(* CoDeSys 2.3 project: esx_ioxp_PPS_load_16.pro *)
(* Libraries: esx_ioxp.lib 19.12.13 13:14:40, Util.lib 18.5.10 15:14:28, Standard.lib 4.10.05 11:14:46 *)

(* PLC configuration (modules and I/O channels)
gq_Ignition AT %IX0.0 [X_SYS_IGNITION] Ignition pin (D+)
gs16_TempBoard AT %IW1 [X_SYS_TEMP_BOARD] System temperature in degree Celsius
gu32_TimeMs AT %ID1 [X_SYS_TIME_MS] System time in ms
gq_StayAlive AT %QX0.0 [X_SYS_STAY_ALIVE] Stay alive mechanism
gq_Relay AT %QX1.0 [X_SYS_RELAY_1] Safety relay
gs32_SensorSupply AT %QD1 [X_SYS_SENSOR_SUPPLY_1] External sensor supply
gs32_IO01 AT %QD2 [InOut] --- Inj 2-1 ----IO01, PIN 9 (PWM H/L, DO, CC, VIN (40V), DIN) {InOut_Type = X_OUT_TYPE_DIGITAL; InOut_FilterConfig = 0; InOut_Circuit1 = X_OUT_CIRCUIT_HIGH_SIDE; InOut_Circuit2 = X_IN_CIRCUIT_NO_PULL_UP; PWM_MaxValue = 10000}
gs32_IO02 AT %QD3 [InOut] ---- Inj 2-2 ---- IO02, PIN 8 (PWM H/L, DO, CC, VIN (40V), DIN) {InOut_Type = X_IN_TYPE_VOLTAGE_40V; InOut_FilterConfig = 0; InOut_Circuit1 = X_IN_CIRCUIT_ACTIVE_HIGH; InOut_Circuit2 = X_IN_CIRCUIT_PULL_UP; PWM_MaxValue = 10000}
gs32_IO03 AT %QD4 [InOut] --- GAS LED BAR  ---  IO03, PIN 7 (PWM H/L, DO, CC, VIN ( {InOut_Type = X_OUT_TYPE_PWM; InOut_FilterConfig = 0; InOut_Circuit1 = X_OUT_CIRCUIT_PUSH_PULL; InOut_Circuit2 = X_IN_CIRCUIT_NO_PULL_UP; PWM_MaxValue = 10000}
gs32_IO04 AT %QD5 [InOut] --- PPS_emul---- IO04, PIN 6 (PWM H/L, DO, CC, VIN (40V), DIN) {InOut_Type = X_OUT_TYPE_PWM; InOut_FilterConfig = 0; InOut_Circuit1 = X_OUT_CIRCUIT_HIGH_SIDE; InOut_Circuit2 = X_IN_CIRCUIT_NO_PULL_UP; PWM_MaxValue = 10000}
gs32_IO05 AT %QD6 [InOut] -----Inj 1-2 ----- IO05, PIN 13 (PWM H, DO, DIN) {InOut_Type = X_OUT_TYPE_DIGITAL; InOut_FilterConfig = 0; InOut_Circuit1 = X_OUT_CIRCUIT_HIGH_SIDE; InOut_Circuit2 = X_IN_CIRCUIT_NO_PULL_UP; PWM_MaxValue = 10000}
gs32_IO06 AT %QD7 [InOut] ---Inj1-1--- IO06, PIN 12 (PWM H, DO, DIN) {InOut_Type = X_OUT_TYPE_DIGITAL; InOut_FilterConfig = 0; InOut_Circuit1 = X_OUT_CIRCUIT_HIGH_SIDE; InOut_Circuit2 = X_IN_CIRCUIT_NO_PULL_UP; PWM_MaxValue = 10000}
gs32_IO07 AT %QD8 [InOut] --- Inj3-1 -----IO07, PIN 11 (PWM H, DO, DIN) {InOut_Type = uninitialized; InOut_FilterConfig = 0; InOut_Circuit1 = X_IN_CIRCUIT_ACTIVE_HIGH; InOut_Circuit2 = X_IN_CIRCUIT_NO_PULL_UP; PWM_MaxValue = 10000}
gs32_IO08 AT %QD9 [InOut] --- Inj 3-2 --  IO08, PIN 10 (PWM H, DO, DIN) {InOut_Type = X_OUT_TYPE_DIGITAL; InOut_FilterConfig = 0; InOut_Circuit1 = X_OUT_CIRCUIT_HIGH_SIDE; InOut_Circuit2 = X_IN_CIRCUIT_NO_PULL_UP; PWM_MaxValue = 10000}
gs32_IO09 AT %ID2 [InOut] --- SPEED --- IO09, PIN 2 (DIN, FIN, IIN) {InOut_Type = X_IN_TYPE_FREQUENCY; InOut_FilterConfig = 0; InOut_Circuit1 = X_OUT_CIRCUIT_HIGH_SIDE; InOut_Circuit2 = X_IN_CIRCUIT_NO_PULL_UP; PWM_MaxValue = 10000}
gs32_IO10 AT %ID3 [InOut] ---RPM--- IO10, PIN 3 (DIN, FIN, IIN) {InOut_Type = X_IN_TYPE_FREQUENCY; InOut_FilterConfig = 0; InOut_Circuit1 = X_IN_CIRCUIT_ACTIVE_HIGH; InOut_Circuit2 = X_IN_CIRCUIT_NO_PULL_UP; PWM_MaxValue = 10000}
gs32_IO11 AT %ID4 [InOut] IO11, PIN 4 (DIN, FIN, IIN) {InOut_Type = uninitialized; InOut_FilterConfig = 0; InOut_Circuit1 = X_IN_CIRCUIT_ACTIVE_HIGH; InOut_Circuit2 = X_IN_CIRCUIT_NO_PULL_UP; PWM_MaxValue = 10000}
gs32_IO12 AT %ID5 [InOut] ---BLOCK ON--- IO12, PIN 5 (DIN) {InOut_Type = X_IN_TYPE_VOLTAGE_10V; InOut_FilterConfig = 0; InOut_Circuit1 = X_IN_CIRCUIT_ACTIVE_HIGH; InOut_Circuit2 = X_IN_CIRCUIT_NO_PULL_UP; PWM_MaxValue = 10000}
gs32_IO13 AT %ID6 [InOut] IO13, PIN 38 (CIN (20mA), DIN) {InOut_Type = uninitialized; InOut_FilterConfig = 0; InOut_Circuit1 = X_IN_CIRCUIT_ACTIVE_HIGH; InOut_Circuit2 = X_IN_CIRCUIT_NO_PULL_UP; PWM_MaxValue = 10000}
gs32_IO14 AT %ID7 [InOut] IIO14, PIN 24 (CIN (20mA), DIN) {InOut_Type = uninitialized; InOut_FilterConfig = 0; InOut_Circuit1 = X_IN_CIRCUIT_ACTIVE_HIGH; InOut_Circuit2 = X_IN_CIRCUIT_NO_PULL_UP; PWM_MaxValue = 20000}
gs32_IO15 AT %ID8 [InOut] - Injecor temp ----IO15, PIN 39 (CIN (20mA), DIN) {InOut_Type = X_IN_TYPE_CURRENT; InOut_FilterConfig = 0; InOut_Circuit1 = X_IN_CIRCUIT_ACTIVE_HIGH; InOut_Circuit2 = X_IN_CIRCUIT_NO_PULL_UP; PWM_MaxValue = 4000000}
gs32_IO16 AT %ID9 [InOut] IO16, PIN 25 (CIN (20mA), DIN) {InOut_Type = uninitialized; InOut_FilterConfig = 0; InOut_Circuit1 = X_IN_CIRCUIT_ACTIVE_HIGH; InOut_Circuit2 = X_IN_CIRCUIT_NO_PULL_UP; PWM_MaxValue = 10000}
gs32_IO17 AT %ID10 [InOut] IO17, PIN 40 (CIN (20mA), DIN) {InOut_Type = uninitialized; InOut_FilterConfig = 0; InOut_Circuit1 = X_IN_CIRCUIT_ACTIVE_HIGH; InOut_Circuit2 = X_IN_CIRCUIT_NO_PULL_UP; PWM_MaxValue = 10000}
gs32_IO18 AT %ID11 [InOut] ----- SOLARKA meter ----- IO18, PIN 26 (CIN (20mA), DIN) {InOut_Type = X_IN_TYPE_CURRENT; InOut_FilterConfig = 0; InOut_Circuit1 = X_IN_CIRCUIT_ACTIVE_HIGH; InOut_Circuit2 = X_IN_CIRCUIT_NO_PULL_UP; PWM_MaxValue = 20000}
gs32_IO19 AT %ID12 [InOut] --- GAS meter  ----- IO19, PIN 41 (CIN (20mA), DIN) {InOut_Type = X_IN_TYPE_CURRENT; InOut_FilterConfig = 0; InOut_Circuit1 = X_IN_CIRCUIT_ACTIVE_HIGH; InOut_Circuit2 = X_IN_CIRCUIT_NO_PULL_UP; PWM_MaxValue = 10000}
gs32_IO20 AT %ID13 [InOut] ---Reductor_temp---  IO20, PIN 27 (CIN (20mA), DIN) {InOut_Type = X_IN_TYPE_CURRENT; InOut_FilterConfig = 0; InOut_Circuit1 = X_IN_CIRCUIT_ACTIVE_HIGH; InOut_Circuit2 = X_IN_CIRCUIT_NO_PULL_UP; PWM_MaxValue = 20000}
gs32_IO21 AT %ID14 [InOut] ---Turbo_pressure--- IO21, PIN 34 (VIN (10V), DIN) {InOut_Type = X_IN_TYPE_VOLTAGE_10V; InOut_FilterConfig = 0; InOut_Circuit1 = X_IN_CIRCUIT_ACTIVE_HIGH; InOut_Circuit2 = X_IN_CIRCUIT_NO_PULL_UP; PWM_MaxValue = 10000}
gs32_IO22 AT %ID15 [InOut] ---Reductor_press---   IO22, PIN 20 (VIN (10V), DIN) {InOut_Type = X_IN_TYPE_VOLTAGE_10V; InOut_FilterConfig = 0; InOut_Circuit1 = X_IN_CIRCUIT_ACTIVE_HIGH; InOut_Circuit2 = X_IN_CIRCUIT_NO_PULL_UP; PWM_MaxValue = 10000}
gs32_IO23 AT %ID16 [InOut] --- EGT ----IO23, PIN 35 (VIN (10V), DIN) {InOut_Type = X_IN_TYPE_VOLTAGE_10V; InOut_FilterConfig = 0; InOut_Circuit1 = X_IN_CIRCUIT_ACTIVE_HIGH; InOut_Circuit2 = X_IN_CIRCUIT_NO_PULL_UP; PWM_MaxValue = 10000}
gs32_IO24 AT %ID17 [InOut] ---PPS1--- IO24, PIN 21 (VIN (10V), DIN) {InOut_Type = X_IN_TYPE_VOLTAGE_10V; InOut_FilterConfig = 0; InOut_Circuit1 = X_IN_CIRCUIT_ACTIVE_HIGH; InOut_Circuit2 = X_IN_CIRCUIT_NO_PULL_UP; PWM_MaxValue = 10000}
gs32_IO25 AT %ID18 [InOut] --- PPS2 ---- IO25, PIN 36 (VIN (10V), DIN) {InOut_Type = X_IN_TYPE_VOLTAGE_10V; InOut_FilterConfig = 0; InOut_Circuit1 = X_IN_CIRCUIT_ACTIVE_HIGH; InOut_Circuit2 = X_IN_CIRCUIT_NO_PULL_UP; PWM_MaxValue = 10000}
gs32_IO26 AT %ID19 [InOut] ---- Check_PPS_emul ----O26, PIN 22 (VIN (10V), DIN) {InOut_Type = X_IN_TYPE_VOLTAGE_10V; InOut_FilterConfig = 0; InOut_Circuit1 = X_IN_CIRCUIT_ACTIVE_LOW; InOut_Circuit2 = X_IN_CIRCUIT_NO_PULL_UP; PWM_MaxValue = 5000}
RS232 [X_SER_1] node 1, in %IB80 out %QB40 {X_SER_BITRATE = 19200; X_SER_STOPBITS = 1; X_SER_MODE = 8 data bits - no parity; X_SER_RX_BUFSIZE = 256; X_SER_TX_BUFSIZE = 256}
CAN1 [X_CAN_BUS_1_XC2] node 2, in %IB80 out %QB40 {X_CAN_BUS_BITRATE = 125000; X_CAN_BUS_11BIT_MASK = 16#7FF; X_CAN_BUS_29BIT_MASK = 16#1FFFFFFF}
TX AT %ID20 [X_CAN_OBJ_HANDLE] CAN object handle
CAN RX Object [X_CAN_OBJ_RX_XC2] node 11770, in %IB84 out %QB40 {X_CAN_OBJ_ID = 16#100; X_CAN_OBJ_XTD = 11bit; X_CAN_OBJ_MASK = 16#7FF; X_CAN_OBJ_SOFT_BUFFER = 10; X_CAN_OBJ_HARD_BUFFER = 10}
  RX AT %ID21 [X_CAN_OBJ_HANDLE] CAN object handle
CAN2 [X_CAN_BUS_2_XC2] node 3, in %IB80 out %QB40 {X_CAN_BUS_BITRATE = 125000; X_CAN_BUS_11BIT_MASK = 16#7FF; X_CAN_BUS_29BIT_MASK = 16#1FFFFFFF}
*)

(* Task configuration *)
TASK Get_RPM (PRIORITY := 3, INTERVAL := T#300ms);
	Get_RPM_speed();
	Get_EGT();
END_TASK
TASK Main (PRIORITY := 20, INTERVAL := T#100ms);
	PLC_PRG();
	DFPRS_Change_Cal_Table();
	Get_Currents();
	Get_Reductor_press();
END_TASK
TASK Act_control (PRIORITY := 2, INTERVAL := T#100ms);
	Act_control();
END_TASK
TASK Get_turbo (PRIORITY := 3, INTERVAL := T#50ms);
	Get_Turbo();
END_TASK
TASK Get_key (PRIORITY := 10, INTERVAL := T#50ms);
	Get_Key();
END_TASK
TASK Get_low_freq (PRIORITY := 5, INTERVAL := T#300ms);
	Get_Gas_meter();
	Get_Reductor_temp();
	Get_Inj_temp();
	Get_FUEL_meter();
	Get_cPPS();
END_TASK
TASK CAN (PRIORITY := 20, INTERVAL := T#50ms);
	Send();
	Recieve();
END_TASK

(* Global variable list: Global_Constant *)
VAR_GLOBAL CONSTANT
(********************** Разное ***************************************************************************)

	TOOTH_NUM					:WORD:=58;				(* Количество зубцов на коленвале *)
	Min_time_cnange_mode_EGT:UDINT:=60000; 		(* Минимальное время в мс между сменами режимов ГАЗ и ДИЗЕЛЬ для обновления статистических значений EGT *)
	Inj_PWM_period				:WORD:=250;				(* Период работы форсунок HANA=16 HZ задается в кол-ве рабочих циклов по 250 мкс*)

(******************** Настойки системы безопасности **********************************)

	RPM_count:WORD:=10;						(* Максимальное количество циклов неправильного RPM, когда считаем это флуктуацией *)
	PPS_err_time:WORD:=3;					(* Максимальное количество циклов неправильного PPS, когда считаем это флуктуацией *)
	Min_Reductor_press_time:WORD:=10;	(* Макстмально допустимое время минимального давления *)
	Reductor_temp_err_time:WORD:=100;	(* Через столько циклов блок опять включится что бы проверить температуру редуктора после первого включения по превышению *)
	EGT_err_time:WORD:=100;					(* Через столько циклов блок опять включится что бы проверить EGT после отключения по превышению EGT *)
	Max_inj_current_time:BYTE:=100;		(* Макстмально допустимое время протекания максимального тока через форсунку в РАБОЧИХ циклах подпрограммы *)

END_VAR

(* Global variable list: Global_Variables *)
VAR_GLOBAL

	(* Значения считывемые с входов контролера *)

	RPM						:WORD; 				(* RPM *)
	Turbo_pressure	      :DINT;				(* Turbo pressure in mV *)
	PPS1	      			:DINT;				(* Основная педаль газа in mV *)
	OLD_PPS					:DINT;
	PPS2						:DINT;				(* Дублирующая педаль газа *)
	EGT						:DINT;				(* Температуры выхлопных газов *)
	Reductor_temp			:DINT;				(* Температура редуктора *)
	Reductor_press			:DINT;				(* Давление после редуктора *)
	Gas_meter				:DINT;				(* Давление газа *)
	Injector_temp			:DINT;				(* Температура инжекторов *)
	FUEL_meter				:DINT;				(* Значение датчика солярки *)
	Speed						:DINT;				(* Счетчик импульсов коленвала *)


	(* РАЗНОЕ *)
	Inj_PWM_time			:BYTE;	 			(* Длительность холдового PWM для газового инжектора, расчитывается исходя из данных калибровки в циклах по 250 мкс*)
	HOLD_time				:BYTE;
	Turn_start				:UDINT;				(* Системное время когда была нажата кнопка управления *)
	Count_min_reductor_press:WORD;			(* Счетчик времени для определения подлинного события падения давления в редукторе *)
	PPS1_emul				:DINT;				(* Уровень PWM для эмулирования первой педали газа *)
	cPPS1_emul				:DINT;				(* Уровень ФАКТИЧЕСКОГО измеренного напряжения эмуляции PPS *)
	FUEL_volume				:REAL;				(* Объем топлива в литрах *)
	Load						:BYTE;				(* Отношение импульсов датчика распредвала и коленвала *)

	(* Значения тока протекающего через Пин, подключеннный к форсунке. 2 Пина = 1 форсунка *)

	s32_Current_Inj1_1			: DINT;
	s32_Current_Inj1_2			: DINT;
	s32_Current_Inj2_1			: DINT;
	s32_Current_Inj2_2			: DINT;
	s32_Current_Inj3_1			: DINT;
	s32_Current_Inj3_2			: DINT;

	(* Структуры данных для записи в EEPROM *)

	p							:Parameters;		(* Сруктура с настройками, при старте контролера подгружаться из EEPROM*)
	a							:Always_write;		(* Структура тоже с настройками. но которая ВСЕГДА при записывается EEPROM при выключении  *)

	(* Логические переменные для включения различных режимов *)

	Flag_ECU_ON				:BOOL;				(* Контроллер включен *)
	Flag_PWM_researh		:BOOL;				(* Включения режима исследования отношения PWM к выходу операционного усилителя *)
	Flag_Inj_PWM_cor		:BOOL;				(* Показывает что была произведена коррекци Inj_PWM по превышению предельных значений *)
	Flag_first_start		:BOOL:=TRUE;		(* Первое включение, для проверки давления *)
	Flag_24V					:BOOL:=FALSE;   	(* 24 Вольтовое газовое оборудоыание, нужен для уменьшения подачи через спецкоды *)

	(* Индивидуальное включение/выключение форсунок *)
	(* Скания все три включены *)
	(* Газель включен первый канал , 2 форсунки. 2 и 3 - выключены  *)
	Flag_Inj1_ON			:BOOL:=TRUE;
	Flag_Inj2_ON			:BOOL:=FALSE;
	Flag_Inj3_ON			:BOOL:=FALSE;

	(* Режим тестирования работы газовых инжекторов *)
	Flag_test_inj: BOOL;

	(* Логические переменные, использующиеся для обмена по CAN калибровками с питоновской прграммой *)

	Flag_CAN_send			:BOOL;				(* Запрос по CAN на посылку калибровки *)
	Flag_CAN_recieve		:BOOL;				(* Запрос по CAN на прием калибровки *)
	Flag_CAN					:BOOL;				(* Режим обмена по CAN калибровками активирован *)
	Flag_CAN_data			:BOOL;
	Flag_CAN_CRC16			:BOOL;
	Flag_CAN_Write			:BOOL;


	(*********** Флаги ошибок  *****************************)

	Err_RPM					:BOOL;				(* RPM более чем RPM_count циклов не в пределах RPM_min - RPM_max *)
	Err_EGT					:BOOL;				(* Превышен максимальный уровень EGT *)
	Err_Reductor_temp		:BOOL;				(* Недостигнута рабочая температура редуктора *)
	Err_Inj1					:BOOL;				(* Долговременно превышен максимальный ток в инжекторе 1 *)
	Err_Inj2					:BOOL;				(* Долговременно превышен максимальный ток в инжекторе 2 *)
	Err_Inj3					:BOOL;				(* Долговременно превышен максимальный ток в инжекторе 3 *)
	Err_Inj_temp			:BOOL;				(* Превышение температуры инжекторов *)
	Err_Reductor_press	:BOOL;				(* Давление в редукторе ниже нормы *)
	Err_PPS					:BOOL;				(* PPS ниже или выше допустимого значения *)

	Can_buffer				:ARRAY [1..6000] OF BYTE; 											(* Буфер для сохранения области EEPROM 750*8 *)

END_VAR

(* Data type *)
(* Эта структурв перезаписывается каждый раз при выключении *)

TYPE Always_write :
STRUCT
		Flag_byte					:BYTE;				(* 8 флагов, для хранения в EEPROM *)
		EGT_max_abs_GAS			:DINT;				(* Абсолютное максимальное достигнутое значение EGT за все время работы контроллера на ГАЗУ *)
		EGT_max_abs_DIESEL		:DINT;				(* Абсолютное максимальное достигнутое значение EGT за все время работы контроллера на ДИЗЕЛЕ *)
		EGT_max_sessions_GAS		:DINT;				(* Абсолютное максимальное значение EGT за прошлую сессию на ДИЗЕЛЕ *)
		EGT_max_sessions_DIESEL	:DINT;				(* Абсолютное максимальное значение EGT за прошлую сессию на ГАЗУ *)
END_STRUCT
END_TYPE

(* Data type *)
TYPE Cal_data :
STRUCT
	Gas: BYTE;
	Diesel: BYTE;
END_STRUCT
END_TYPE

(* Data type *)
(* Используется для обхода ограничений по редактированию таблиц в визуализации *)

TYPE FLS :
STRUCT
	a:WORD;
END_STRUCT
END_TYPE

(* Data type *)
(* Структура данных, хранящаяся в EEPROM *)
TYPE Parameters :
	STRUCT
		(* Таблица для 3-х мерной калибровки подачи газа и дизеля. Оброты, надув, педаль ( разносится автоматически ) *)
		Cal_table					:ARRAY [1..16,1..16] OF Cal_data;
		(* Основные таблицы границ  - обротов, надува и педали газа *)
		RPM_table					:ARRAY[1..16] OF WORD;	(* Значения RPM *)
		Turbo_table					:ARRAY[1..16] OF WORD;	(* Значения наддува турбины *)
		PPS_table					:ARRAY[1..16] OF WORD;	(* Значения нажатия на педаль газа *)
		PPS1_emul_PWM				:ARRAY[1..32] OF WORD;	(* Соответствие значения эмуляции и частотв PWM *)
		(* Учет топлива *)
		LED_BAR_PWM					:ARRAY[1..5]  OF WORD;	(* Соответствие PWM каждому диапазону датчика давления для индикатора *)
		Gas_meter_volume			:ARRAY[1..5]  OF DINT;	(* Разбивка датчика давления в баллоне на диапазоны *)
		FUEL_meter_dat				:ARRAY[1..32] OF WORD;	(* Калибровка датчика солярки, соответствие показаний физическому объему, показания датчика *)
		FUEL_meter_liter			:ARRAY[1..32] OF WORD;	(* Калибровка датчика литры *)
		(******************** Настойки системы безопасности **********************************)
		EGT_max						:WORD;						(* Максимально допустимый уровень EGT *)
		(*********** Пределы допустимых значений RPM ******************************)
		RPM_Min						:WORD;						(* Минимальный порог допкстимого RPM *)
		RPM_Max						:WORD;						(* Максимальный порог допустимого RPM *)
		(*********** Пределы допустимых для редуктора ******************************)
		Reductor_temp_work		:WORD;						(* Минимальная температура редуктора для включения блока *)
		Min_Reductor_press		:WORD;						(* Минимальное давление редуктора для включения блока *)
		(*********** Пределы допустимых для педали газа ******************************)
		PPS1_min						:WORD;						(* Минимальный порог для PPS *)
		PPS1_max						:WORD;						(* Максимальный порог для PPS *)
		PPS2_min						:WORD;						(* Минимальный порог для PPS *)
		PPS2_max						:WORD;						(* Максимальный порог для PPS *)
		PPS_ratio_min				:REAL;						(* Минимальный корректный порог соотношений значений PPS1 и PPS2 *)
		PPS_ratio_max				:REAL;						(* Максимальный корректный порог соотношений значений PPS1 и PPS2 *)
		(**************** Управление форсунками ***************************************************************************)
		Inj_Low_period				:WORD;						(* Задание скважности PWM форсунок (соотношение кол-ва ЦИКЛОВ низкого сигнала к одному ВЫСОКОМУ циклу), подбирается имперически по условию соблюдения уровня холдового тока на форсунке *)
		Inj_High_period			:WORD;						(* Задание скважности PWM форсунок (соотношение кол-ва ЦИКЛОВ низкого сигнала к одному ВЫСОКОМУ циклу), подбирается имперически по условию соблюдения уровня холдового тока на форсунке *)
		Inj_MAX_hold_time			:BYTE;						(* В циклах по 250 мкс !Максимально возможная длительность холда для форсунок на больших нагрузках *)
		Inj_MAX_hold_time_min	:BYTE;						(* Максимально возможная длительность холда для форсунок на малых нагрузках *)
		Inj_peak_curent_cycle	:BYTE;						(* Количество срабатываний цикла обработчика прерываний, для генерирования импульса длительности открытия форсунки с пиковым током в циклах по 250 мкс*)
		(* SCANIA P380 -  Максимальная температура форсунок 90 C при балластном резисторе 1050 Ом  4325 *)
		(* Газель - Максимальная температура форсунок 110 C при балластном резисторе 560 Ом* это 16000, но так как температура растет очень медленно то для подстраховки ставим 14000*)
		Inj_temp_max				:DINT;
		Max_inj_current			:DWORD;						(* Максимальный длительный ток через газовые форсунки в микроамперах *)
		Min_inj_current			:DWORD;						(* Минимальный длительный ток ( обрыв ) через газовые форсунки в микроамперах *)

		Speed_limit					:WORD;						(* Минимальная скорость с какой начинать подачу газа и эмуляцию *)
		Load_table					:ARRAY[1..16] OF WORD;	(* Значения нажатия на педаль газа *)
		GAS_Load_table				:ARRAY[1..16] OF INT;	(* Значения нажатия на педаль газа *)
		DIESEL_Load_table			:ARRAY[1..16] OF INT;	(* Значения нажатия на педаль газа *)
	END_STRUCT
END_TYPE

(* POU Ввод данных/Get_RPM_speed, ST *)
PROGRAM Get_RPM_speed
VAR

	s16_Return   		: INT;
   Old_pulse_counter, Pulse_counter,s32_Counter    	: DINT; (* Набор переменных для вычисления RPM *)
	Old_pulse_counter_speed,s32_Counter_speed    	: DINT; (* Набор переменных для вычисления оборотов коленвала *)
   fb_InGetCounter   : FB_x_in_get_counter;

	cycle_time: DINT;
	old_time: DINT;
	Flag_speed_OK:BOOL;				(* Флаг для визуализации *)
	i: WORD:=RPM_count;			(* Для начала работы нужно хоть одно правильное значение RPM *)
END_VAR
(* Получаем количество импульсов ( импульс=2 сигнала=открывающий и закрывающий фронт )с датчика Холла *)
fb_InGetCounter(ou16_Channel:=X_IN_10, os32_Value=>s32_Counter, os16_Status=>s16_Return);
(* Вычисляем количество импульсов за цикл работы этой прграммы *)
Pulse_counter:=s32_Counter-old_pulse_counter;
Old_pulse_counter:=s32_Counter;
(* Вычисляем время цикла в ms*)
cycle_time:=gu32_TimeMs-old_time;
old_time:=gu32_TimeMs;
(* Переводим в RPM с учетом отсутствующих зубов и времени цикла 30000=1000*60/2 *)
RPM:=DINT_TO_WORD((Pulse_counter*30000/cycle_time)/TOOTH_NUM);
Check_RPM();

(* Получаем количество импульсов ( импульс=2 сигнала=открывающий и закрывающий фронт )с датчика Холла *)
fb_InGetCounter(ou16_Channel:=X_IN_09, os32_Value=>s32_Counter_speed, os16_Status=>s16_Return);
(* Вычисляем количество импульсов за цикл работы этой прграммы *)
Speed:=s32_Counter_speed-old_pulse_counter_speed;
Old_pulse_counter_speed:=s32_Counter_speed;
(* Соотношение между оборотами двигателя и оборотами коленвала *)
IF Speed <> 0 THEN
	Load:=DINT_TO_BYTE(Pulse_counter/Speed);
ELSE
	Load:=0;
END_IF
(* Для визуализации *)
IF speed > p.Speed_limit THEN
	Flag_speed_OK:=TRUE;
ELSE
	Flag_speed_OK:=FALSE;
END_IF
END_PROGRAM
ACTION Check_RPM:
(* Находится ли RPM в допустимых пределах ? *)
IF RPM < p.RPM_min OR RPM > p.RPM_max THEN
	i:=i+1;
ELSE
	i:=0;
END_IF
(* Если RPM выходит задопустимые пределы RPM_count раз подряд, тогда ошибка *)
IF i>=RPM_count THEN
	Err_RPM:=TRUE;
	i:=RPM_count;					(* Что бы избежать переполнения и ложного сброса флага *)
ELSE
	Err_RPM:=FALSE;
END_IF
END_ACTION

(* POU Ввод данных/Get_EGT, ST *)
PROGRAM Get_EGT
VAR
	fb_InGetValue   : FB_x_in_get_value;
	s16_Return      : INT;
	EGT_err_flag: BOOL; (* EGT уже больше, но пока время для установления главного флага еще не вышло *)
	Count_max_EGT: WORD;
	Flag_EGT_reset: BOOL;
END_VAR
fb_InGetValue(ou16_Channel:=X_IN_23, os32_Value=>EGT, os16_Status=>s16_Return);

(* Если EGT превысило допустимую температуру, то следующий контроль EGT на возможное включение блока произойдет через некоторое время *)

IF EGT_err_flag AND  Count_max_EGT < EGT_err_time THEN
	Count_max_EGT:=Count_max_EGT+1;
ELSE
	Count_max_EGT:=0;
	(* Находится ли EGT в допустимых пределах ? *)
	IF EGT > p.EGT_max THEN
		EGT_err_flag:=TRUE;
		Err_EGT:=TRUE;
	ELSE
		EGT_err_flag:=FALSE;
		Err_EGT:=FALSE;
	END_IF
END_IF

(* Контроль, что бы между сменами режимов прошло достаточно кол-ва времени *)
IF (gu32_TimeMs-Turn_start) > Min_time_cnange_mode_EGT THEN
(* Запись максимального значения EGT в как течении сесии так и абсолютно за все время *)
		IF Flag_ECU_ON THEN
				IF EGT > a.EGT_max_sessions_GAS	THEN
					a.EGT_max_sessions_GAS:=EGT;
				END_IF
				IF EGT > a.EGT_max_abs_GAS	THEN
					a.EGT_max_abs_GAS:=EGT;
				END_IF
		ELSE
				IF EGT > a.EGT_max_sessions_DIESEL	THEN
					a.EGT_max_sessions_DIESEL:=EGT;
				END_IF
				IF EGT > a.EGT_max_abs_DIESEL	THEN
					a.EGT_max_abs_DIESEL:=EGT;
				END_IF
		END_IF
END_IF

(* Если нажата кнопка RESET в визуализации, то сбрасываем все значения в структуре always_write где хранятся байт флагов и значения EGT *)
IF Flag_EGT_reset THEN
	a.EGT_max_abs_GAS:=0;
	a.EGT_max_abs_DIESEL:=0;
	a.EGT_max_sessions_GAS:=0;
	a.EGT_max_sessions_DIESEL:=0;
	Flag_EGT_reset:=FALSE;
END_IF
END_PROGRAM

(* POU PLC_PRG, ST *)
PROGRAM PLC_PRG
VAR
	q_FirstCycle	: BOOL := TRUE;

	fb_SysClose		: FB_x_sys_close;
	fb_SsvTrigger	: FB_x_ssv_trigger;
	s16_Return,s16_Return3		: INT;

(*  Работа с входами *)
	fb_InInit    	: FB_x_in_init;
(* Работы с выходами *)
	fb_OutInit  	: FB_x_out_init;
	fb_OutSetFrequency   : FB_x_out_set_frequency;
	fb_OutSetValue   : FB_x_out_set_value;
(* Работа с таймером *)
   fb_TimClose   : FB_x_tim_close;
   fb_TimInit    : FB_x_tim_init;
   fb_TimSet     : FB_x_tim_set;
(* Работа с энергонезависимой памятью *)
	fb_EepWrite   	: FB_x_eep_write;
	fb_EepRead  	: FB_x_eep_read;

	i,k,z								:BYTE;				(* Служат для формирования байта флагов *)

	EGT_max_prev_sessions_GAS		:DINT;				(* Абсолютное максимальное значение EGT за прошлую сессию на ДИЗЕЛЕ *)
	EGT_max_prev_sessions_DIESEL	:DINT;				(* Абсолютное максимальное значение EGT за прошлую сессию на ГАЗУ *)

	Count_off: BYTE;
END_VAR
IF (q_FirstCycle = TRUE) THEN
	q_FirstCycle := FALSE;
	(* deactivate 'Safety relay' *)
	gq_Relay := FALSE;
	(* activate 'Stay alive' mechanism *)
	gq_StayAlive := TRUE;
	(* activate 'Sensor Supply' *)
	gs32_SensorSupply := X_SYS_SENSOR_SUPPLY_10V;

	Read_EEPROM();				(* Инициализируем переменные значениями из EEPROMa *)
	Init_IN();					(* Инициализируем входы *)
	Init_OUT();					(* Инициализируем выходы *)
	Init_timer();				(* Инициализируем таймер *)

	Turn_start:=gu32_TimeMs;(* Для организации паузы при включении для лога EGT *)

	(* Сохраняем значения счетчиков в целях индикации *)
	EGT_max_prev_sessions_GAS:=a.EGT_max_sessions_GAS;
	EGT_max_prev_sessions_DIESEL:=a.EGT_max_sessions_DIESEL;
	(* Для расчета максимальныйх значений именно в текущей сессии обнуляем счетчики *)
	a.EGT_max_sessions_GAS:=0;
	a.EGT_max_sessions_DIESEL:=0;

END_IF
(* trigger 'System Supervisor' *)
fb_SsvTrigger(ou16_TriggerType:=X_SSV_TRIGGER);

Check_ON();			(* Проверка стратовых условий *)

IF (gq_Ignition = FALSE) THEN
	(* Ignition (D+) was switched off *)
	fb_TimClose(ou32_Handle:=fb_TimInit.ou32_Handle);
	(* Запакрвываем флаги в байт *)
	a.Flag_byte:=PACK(B0:=0,B1:=0,B2:=0,B3:=0,B4:=0,B5:=0,B6:=Flag_CAN,B7:=Flag_ECU_ON);
	(* Записывем параметры газодизельного блока в энергонезависимую память *)
	fb_EepWrite(ou32_Address:=SIZEOF(p), ou32_Count:=SIZEOF(a), opu8_Data:=ADR(a), os16_Status=>s16_Return);
	(* close ESX-IOXp properly *)
	fb_SysClose();
END_IF
END_PROGRAM
ACTION Check_ON:
(* Проверка стратовых условий *)
IF Flag_ECU_ON THEN											(* В любом случае кнопка отключает все *)
		IF Flag_test_inj OR Flag_PWM_researh THEN		(* Есть ли спецрежимы отладки в которых проверка наличий условий для работы не производится ?*)
				gq_Relay := TRUE;									(* Главное реде ВКЛ  activate 'Safety relay'*)
		ELSE
		(* Если все условия выполняются включаем главное реле *)
				IF Err_RPM=FALSE AND Err_EGT=FALSE AND Err_Reductor_temp=FALSE AND Err_Inj1=FALSE AND
 				Err_inj2=FALSE AND Err_inj3=FALSE AND Err_inj_temp=FALSE AND Err_PPS=FALSE THEN
						IF Flag_first_start THEN								(* Спец режим тестового включения отсечного клапана при первом старте *)
								gq_Relay := TRUE;									(* Главное реде ВКЛ  activate 'Safety relay'*)
								Flag_first_start:= FALSE;
						ELSIF Err_Reductor_press=FALSE THEN
								gq_Relay := TRUE;									(* Главное реде ВКЛ  activate 'Safety relay'*)
						ELSE
								gq_Relay := FALSE;								(* Главное реде ВЫКЛ  deactivate 'Safety relay'*)
						END_IF
				ELSE
						gq_Relay := FALSE;	(* Главное реде ВЫКЛ  deactivate 'Safety relay'*)
				END_IF
		END_IF
ELSE
		gq_Relay := FALSE;								(* Главное реде ВЫКЛ  deactivate 'Safety relay'*)
END_IF
END_ACTION
ACTION Init_IN:
(**************** ИНИЦИАЛИЗАЦИЯ ВХОДОВ **************************)

(********************** Замер частоты *****************************)

(* Инициализируем вход 10, пин 3 как RPM вход *)
fb_InInit(	ou16_Channel:=X_IN_10,
        		ou16_Type:=X_IN_TYPE_FREQUENCY,
         	ou16_FilterConfig:=0,
	         ou16_InputCircuit:=X_IN_CIRCUIT_ACTIVE_HIGH,
          	ou32_CallbackParameter:=0,
	         ou16_EventCallback:=0,
          	os16_Status=>s16_Return);

(* Инициализируем вход 10, пин 2 как вход c датчика скорости *)
fb_InInit(	ou16_Channel:=X_IN_09,
        		ou16_Type:=X_IN_TYPE_FREQUENCY,
         	ou16_FilterConfig:=0,
	         ou16_InputCircuit:=X_IN_CIRCUIT_ACTIVE_HIGH,
          	ou32_CallbackParameter:=0,
	         ou16_EventCallback:=0,
          	os16_Status=>s16_Return);

(*********** Цифровой вход ********************************************)

(* Инициализируем вход 12, пин 5 как дискретный вход включения газодизельного блока  *)
fb_InInit(	ou16_Channel:=X_IN_12,
        		ou16_Type:=X_IN_TYPE_DIGITAL,
         	ou16_FilterConfig:=0,
	         ou16_InputCircuit:=X_IN_CIRCUIT_ACTIVE_HIGH,
          	ou32_CallbackParameter:=0,
	         ou16_EventCallback:=0,
          	os16_Status=>s16_Return);

(****************** Замер напряжения *****************************************)

(************************************* PPS **********************************************)

(* Инициализируем вход 24, пин 21 как вход 0..10V для основной педали газа PPS1 в mV *)
fb_InInit(	ou16_Channel:=X_IN_24,
        		ou16_Type:=X_IN_TYPE_VOLTAGE_10V,
         	ou16_FilterConfig:=0,
	         ou16_InputCircuit:=X_IN_CIRCUIT_ACTIVE_HIGH,
          	ou32_CallbackParameter:=0,
	         ou16_EventCallback:=0,
          	os16_Status=>s16_Return);

(* Инициализируем вход 25, пин 36 как вход 0..10V для PPS 2 *)
fb_InInit(	ou16_Channel:=X_IN_25,
        		ou16_Type:=X_IN_TYPE_VOLTAGE_10V,
         	ou16_FilterConfig:=0,
	         ou16_InputCircuit:=X_IN_CIRCUIT_ACTIVE_HIGH,
          	ou32_CallbackParameter:=0,
	         ou16_EventCallback:=0,
          	os16_Status=>s16_Return);

(*****************************************************************************************)

(* Инициализируем вход 21, пин 34 как вход 0..10V для Turbo pressure в mV *)
fb_InInit(	ou16_Channel:=X_IN_21,
        		ou16_Type:=X_IN_TYPE_VOLTAGE_10V,
         	ou16_FilterConfig:=0,
	         ou16_InputCircuit:=X_IN_CIRCUIT_ACTIVE_HIGH,
          	ou32_CallbackParameter:=0,
	         ou16_EventCallback:=0,
          	os16_Status=>s16_Return);


(* Инициализируем вход 22, пин 20 как вход 0..10V для Reductor press в mV *)
fb_InInit(	ou16_Channel:=X_IN_22,
        		ou16_Type:=X_IN_TYPE_VOLTAGE_10V,
         	ou16_FilterConfig:=0,
	         ou16_InputCircuit:=X_IN_CIRCUIT_ACTIVE_HIGH,
          	ou32_CallbackParameter:=0,
	         ou16_EventCallback:=0,
          	os16_Status=>s16_Return);

(* Инициализируем вход 23, пин 35 как вход 0..10V для EGT в mV *)
fb_InInit(	ou16_Channel:=X_IN_23,
        		ou16_Type:=X_IN_TYPE_VOLTAGE_10V,
         	ou16_FilterConfig:=0,
	         ou16_InputCircuit:=X_IN_CIRCUIT_ACTIVE_HIGH,
          	ou32_CallbackParameter:=0,
	         ou16_EventCallback:=0,
          	os16_Status=>s16_Return);

(* Инициализируем вход 26 , пин 22 как вход 0..10V для контроля выдачи эмуляции PPS *)
fb_InInit(	ou16_Channel:=X_IN_26,
        		ou16_Type:=X_IN_TYPE_VOLTAGE_10V,
         	ou16_FilterConfig:=0,
	         ou16_InputCircuit:=X_IN_CIRCUIT_ACTIVE_HIGH,
          	ou32_CallbackParameter:=0,
	         ou16_EventCallback:=0,
          	os16_Status=>s16_Return);

(**************** Замер тока *******************************)

(* Инициализируем вход 19, пин 41 как токовый вход для датчика давления газа  *)
fb_InInit(	ou16_Channel:=X_IN_19,
        		ou16_Type:=X_IN_TYPE_CURRENT,
         	ou16_FilterConfig:=0,
	         ou16_InputCircuit:=X_IN_CIRCUIT_ACTIVE_HIGH,
          	ou32_CallbackParameter:=0,
	         ou16_EventCallback:=0,
          	os16_Status=>s16_Return);

(* Инициализируем вход 20, пин 27 как токовый вход для датчика температуры редуктора  *)
fb_InInit(	ou16_Channel:=X_IN_20,
        		ou16_Type:=X_IN_TYPE_CURRENT,
         	ou16_FilterConfig:=0,
	         ou16_InputCircuit:=X_IN_CIRCUIT_ACTIVE_HIGH,
          	ou32_CallbackParameter:=0,
	         ou16_EventCallback:=0,
          	os16_Status=>s16_Return);

(* Инициализируем вход 15, пин 39 как токовый вход для датчика температуры инжекторов  *)
fb_InInit(	ou16_Channel:=X_IN_15,
        		ou16_Type:=X_IN_TYPE_CURRENT,
         	ou16_FilterConfig:=0,
	         ou16_InputCircuit:=X_IN_CIRCUIT_ACTIVE_HIGH,
          	ou32_CallbackParameter:=0,
	         ou16_EventCallback:=0,
          	os16_Status=>s16_Return);

(* Инициализируем вход 18, пин 26 как токовый вход для датчика топлива  *)
fb_InInit(	ou16_Channel:=X_IN_18,
        		ou16_Type:=X_IN_TYPE_CURRENT,
         	ou16_FilterConfig:=0,
	         ou16_InputCircuit:=X_IN_CIRCUIT_ACTIVE_HIGH,
          	ou32_CallbackParameter:=0,
	         ou16_EventCallback:=0,
          	os16_Status=>s16_Return);
END_ACTION
ACTION Init_OUT:
(**************** ИНИЦИАЛИЗАЦИЯ ВЫХОДОВ **************************)

(* *************************  ГРУППА ВЫХОДОВ 1 **********************************************************)

(* Инициализируем выход 1, пин 9 как выход управления Инжектором_2-1 *)
fb_OutInit(ou16_Channel:=X_OUT_01,
           ou16_Type:=X_OUT_TYPE_DIGITAL + X_OUT_CIRCUIT_HIGH_SIDE ,
           os32_MaxValue:=1,
           ou32_CallbackParameter:=0,
           ou16_ErrorCallback:=0,
           os16_Status=>s16_Return);

(* Инициализируем выход 1, пин 8 как выход управления Инжектором_2-2 *)
fb_OutInit(ou16_Channel:=X_OUT_02,
           ou16_Type:=X_OUT_TYPE_DIGITAL + X_OUT_CIRCUIT_HIGH_SIDE ,
           os32_MaxValue:=1,
           ou32_CallbackParameter:=0,
           ou16_ErrorCallback:=0,
           os16_Status=>s16_Return);

(* Инициализируем выход 3, пин 7 как выход для выдачи LED *)
fb_OutInit(ou16_Channel:=X_OUT_03,
           ou16_Type:=X_OUT_TYPE_PWM +  X_OUT_CIRCUIT_HIGH_SIDE ,
           os32_MaxValue:=10000,
           ou32_CallbackParameter:=00,
           ou16_ErrorCallback:=0,
           os16_Status=>s16_Return);

(* Инициализируем выход 4, пин 6 как выход для выдачи PPS emul *)
fb_OutInit(ou16_Channel:=X_OUT_04,
           ou16_Type:=X_OUT_TYPE_PWM +  X_OUT_CIRCUIT_HIGH_SIDE ,
           os32_MaxValue:=10000,
           ou32_CallbackParameter:=00,
           ou16_ErrorCallback:=0,
           os16_Status=>s16_Return);

(* *************************  ГРУППА ВЫХОДОВ 2 *********************************************************)

(* Инициализируем выход 5, пин 13 как выход управления Инжектором 1-2 *)
fb_OutInit(ou16_Channel:=X_OUT_05,
           ou16_Type:=X_OUT_TYPE_DIGITAL + X_OUT_CIRCUIT_HIGH_SIDE ,
           os32_MaxValue:=1,
           ou32_CallbackParameter:=0,
           ou16_ErrorCallback:=0,
           os16_Status=>s16_Return);

(* Инициализируем выход 6, пин 12 как выход управления Инжектором 1-1 *)
fb_OutInit(ou16_Channel:=X_OUT_06,
           ou16_Type:=X_OUT_TYPE_DIGITAL + X_OUT_CIRCUIT_HIGH_SIDE ,
           os32_MaxValue:=1,
           ou32_CallbackParameter:=0,
           ou16_ErrorCallback:=0,
           os16_Status=>s16_Return);

(* Инициализируем выход 7, пин 11 как выход управления Инжектором 3-1 *)
fb_OutInit(ou16_Channel:=X_OUT_07,
           ou16_Type:=X_OUT_TYPE_DIGITAL + X_OUT_CIRCUIT_HIGH_SIDE,
           os32_MaxValue:=1,
           ou32_CallbackParameter:=0,
           ou16_ErrorCallback:=0,
           os16_Status=>s16_Return);

(* Инициализируем выход 8, пин 10 как выход управления Инжектором 3-2 *)
fb_OutInit(ou16_Channel:=X_OUT_08,
           ou16_Type:=X_OUT_TYPE_DIGITAL + X_OUT_CIRCUIT_HIGH_SIDE ,
           os32_MaxValue:=1,
           ou32_CallbackParameter:=0,
           ou16_ErrorCallback:=0,
           os16_Status=>s16_Return);
END_ACTION
ACTION Init_TIMER:
(* initialize timer *)

fb_TimInit.ou16_Priority          := X_TIM_PRIO_01;
fb_TimInit.ou32_CallbackParameter := 0;
fb_TimInit.ou16_TimerCallback     := INDEXOF(TimerCallback);
fb_TimInit();
IF (fb_TimInit.os16_Status = C_NO_ERR) THEN      (* set timer *)
		fb_TimSet.ou32_Handle := fb_TimInit.ou32_Handle;
  		fb_TimSet.ou32_DelayTime := 0;
   	fb_TimSet.ou32_CycleTime := 1;
		fb_TimSet();
END_IF
END_ACTION
ACTION Read_EEPROM:
(* Читаем все параметры из энергонезависимой памяти *)
fb_EepRead(ou32_Address:=0, ou32_Count:=SIZEOF(p), opu8_Data:=ADR(p), os16_Status=>s16_Return);
fb_EepRead(ou32_Address:=SIZEOF(p), ou32_Count:=SIZEOF(a), opu8_Data:=ADR(a), os16_Status=>s16_Return);

(* Устанавливаем значение переменных, согласно битам в байте флагов *)

Flag_ECU_ON					:=EXTRACT( X:=a.Flag_byte,N:=7);				(* Биты нумеруются с 0 ! *)
Flag_CAN						:=EXTRACT( X:=a.Flag_byte,N:=6);
END_ACTION

(* POU TimerCallback, ST *)
PROGRAM TimerCallback
VAR
	fb_OutGetCurrent   : FB_x_out_get_current;

	fb_OutSetValue	: FB_x_out_set_value;
	s16_Return   	: INT;
	out				: DINT;  (* Задает уровень выходов *)

	Peak_curent_flag: BOOL:=TRUE;	(* Флаг показывающий, что выполняется выдача пикового тока на форсунки *)
	Peak_curent_counter: WORD;		(* Счетчик циклов выдачи пикового тока на форсунки *)

	Hold_curent_low_counter:WORD;		(* Счетчик циклов выдачи низкого уровня в цикле выдачи холдового тока на форсунки *)
	Hold_curent_High_counter: WORD;

	Hold_curent_counter:WORD;			(* Счетчик циклов выдачи холдового тока на форсунки *)
	Hold_curent_flag: BOOL;				(* Флаг показывающий, что выполняется выдача тока удержаня на газовые форсунки *)

	Inj_Big_cycle: WORD; 				(* Счетчик выполненных циклов в  большом цикле работы форсунок HANA=10 Hz *)
	Inj_hold_High_flag: BOOL;

	Act_PWM_High_flag: BOOL;
	Act_PWM_High_counter: WORD;
	Act_PWM_Low_counter: WORD;

END_VAR
(* Эта програма POU вызывается по таймеру *)

Get_Inj_current(); (* Считываем значения фактического тока с форсунок *)

(* Форсунки фключаются только когда газ и блок включены и имеется холд ток иили включен режим тестирования работы форсунок *)
IF (Flag_ECU_ON AND Inj_PWM_time > 0 AND Speed > p.Speed_limit ) OR Flag_test_inj THEN
				IF Inj_Big_cycle<Inj_PWM_period THEN			(* Большой цикл работы форсунок, длительность которого  Inj_PWM_period установлена производителем. куда входит пиковый ток, холд ток и пауза *)
						Inj_Big_cycle:=Inj_Big_cycle+1;
						(* Выдача пикового тока *)
						IF Peak_curent_flag=TRUE THEN
								IF Peak_curent_counter< p.Inj_peak_curent_cycle THEN (*  Длительность выдачи пикового тока на форсунки Inj_peak_curent_cycle устанавливается производителем задается в разделе констант*)
										Peak_curent_counter:=Peak_curent_counter+1;
										out:=1;
								ELSE
										Peak_curent_counter:=0;
										out:=0;
										Peak_curent_flag:=FALSE;
								END_IF
						ELSIF Hold_curent_flag=TRUE THEN
								(********** Выдача тока удержания *)
								IF Hold_curent_counter<Inj_PWM_time THEN                (* Длительность выдачи тока удержания Inj_PWM_time, выраженная в кол-ве циклов обработчика прерывания вычисляется из данных  калибровочной таблицы *)
										Hold_curent_counter:=Hold_curent_counter+1;
										IF Inj_hold_High_flag=TRUE THEN									(*  Идет генерация импульса высокого уровня *)
												IF Hold_curent_High_counter < p.Inj_High_period THEN
														Hold_curent_High_counter:=Hold_curent_High_counter+1;
														out:=1;
												ELSE
														out:=0;
														Inj_hold_High_flag:=FALSE;
														Hold_curent_Low_counter:=1;
												END_IF
										ELSE																	(* Идет генерация пауз между имплусами высокого уровня *)
												IF Hold_curent_Low_counter < p.Inj_Low_period THEN
														Hold_curent_Low_counter:=Hold_curent_Low_counter+1;
														out:=0;
												ELSE
														Inj_hold_High_flag:=TRUE;
														Hold_curent_High_counter:=1;
														out:=1;
												END_IF
										END_IF
								ELSE
										Hold_curent_counter:=0;
										Hold_curent_flag:=FALSE;
										out:=0;
								END_IF
						END_IF
				ELSE
						Inj_Big_cycle:=0;
						Peak_curent_flag:=TRUE;
						Hold_curent_flag:=TRUE;
				END_IF
		(* Inj 1 *)
		IF Flag_Inj1_ON THEN
			fb_OutSetValue(ou16_Channel:=X_OUT_05, os32_Value:=out, os16_Status=>s16_Return);
			fb_OutSetValue(ou16_Channel:=X_OUT_06, os32_Value:=out, os16_Status=>s16_Return);
		ELSE
			fb_OutSetValue(ou16_Channel:=X_OUT_05, os32_Value:=0, os16_Status=>s16_Return);
			fb_OutSetValue(ou16_Channel:=X_OUT_06, os32_Value:=0, os16_Status=>s16_Return);
		END_IF
		(* Inj 2 *)
		IF Flag_Inj2_ON THEN
			fb_OutSetValue(ou16_Channel:=X_OUT_01, os32_Value:=out, os16_Status=>s16_Return);
			fb_OutSetValue(ou16_Channel:=X_OUT_02, os32_Value:=out, os16_Status=>s16_Return);
		ELSE
			fb_OutSetValue(ou16_Channel:=X_OUT_01, os32_Value:=0, os16_Status=>s16_Return);
			fb_OutSetValue(ou16_Channel:=X_OUT_02, os32_Value:=0, os16_Status=>s16_Return);
		END_IF
		(* Inj 3 *)
		IF Flag_Inj3_ON THEN
			fb_OutSetValue(ou16_Channel:=X_OUT_07, os32_Value:=out, os16_Status=>s16_Return);
			fb_OutSetValue(ou16_Channel:=X_OUT_08, os32_Value:=out, os16_Status=>s16_Return);
		ELSE
			fb_OutSetValue(ou16_Channel:=X_OUT_07, os32_Value:=0, os16_Status=>s16_Return);
			fb_OutSetValue(ou16_Channel:=X_OUT_08, os32_Value:=0, os16_Status=>s16_Return);
		END_IF
ELSE
		(* На всякий случай явно выключим инжекторы, если не выполняются условия их включения *)
		fb_OutSetValue(ou16_Channel:=X_OUT_05, os32_Value:=0, os16_Status=>s16_Return);
		fb_OutSetValue(ou16_Channel:=X_OUT_06, os32_Value:=0, os16_Status=>s16_Return);

		fb_OutSetValue(ou16_Channel:=X_OUT_01, os32_Value:=0, os16_Status=>s16_Return);
		fb_OutSetValue(ou16_Channel:=X_OUT_02, os32_Value:=0, os16_Status=>s16_Return);

		fb_OutSetValue(ou16_Channel:=X_OUT_07, os32_Value:=0, os16_Status=>s16_Return);
		fb_OutSetValue(ou16_Channel:=X_OUT_08, os32_Value:=0, os16_Status=>s16_Return);
END_IF
END_PROGRAM
ACTION Get_Inj_current:
(* Считываем значения фактического тока с форсунок *)

(* Inj1 *)
fb_OutGetCurrent(ou16_Channel:=X_OUT_06, os32_Current=>s32_Current_Inj1_1, os16_Status=>s16_Return);
fb_OutGetCurrent(ou16_Channel:=X_OUT_05, os32_Current=>s32_Current_Inj1_2, os16_Status=>s16_Return);
(* Inj 2 *)
fb_OutGetCurrent(ou16_Channel:=X_OUT_01, os32_Current=>s32_Current_Inj2_1, os16_Status=>s16_Return);
fb_OutGetCurrent(ou16_Channel:=X_OUT_02, os32_Current=>s32_Current_Inj2_2, os16_Status=>s16_Return);
(* Inj 3 *)
fb_OutGetCurrent(ou16_Channel:=X_OUT_07, os32_Current=>s32_Current_Inj3_1, os16_Status=>s16_Return);
fb_OutGetCurrent(ou16_Channel:=X_OUT_08, os32_Current=>s32_Current_Inj3_2, os16_Status=>s16_Return);
END_ACTION

(* POU DFPRS_Change_Cal_Table, ST *)
PROGRAM DFPRS_Change_Cal_Table
VAR
	(* Флаги для инициализации различных действий из визуализации *)
	(* для всей таблицы *)
	Write_cal, Read_cal	:BOOL; (* Считать или записать данные в EEPROM *)
	Write_cal2,Red_cal2	:BOOL; (* Считать или записать данные из таблицы в окно редактора *)
	HALF_set_ALL,Set_ALL,Set_ALL_bufer,Calculate	:BOOL;
	Diagonal_1, Diagonal_2, Diagonal_3, Diagonal_21, Diagonal_31,Diagonal_32: BOOL; (* Флаги для начала обработки диагональных калибровок *)
	ALL_plus, ALL_minus	:BOOL;
	Flag_cal_table_gas	:BOOL; (* Выбор работы с газовой или дизельнгой калибровкой *)
	Fuel_type				:STRING; (* Показывает в визуализации тип калибровки *)


	(* для RPM *)
	RPM_Flag_plus_1,RPM_Flag_plus_2,RPM_Flag_plus_3,RPM_Flag_plus_4,RPM_Flag_plus_5,RPM_Flag_plus_6,RPM_Flag_plus_7,RPM_Flag_plus_8:BOOL;
	RPM_Flag_plus_9,RPM_Flag_plus_10,RPM_Flag_plus_11,RPM_Flag_plus_12,RPM_Flag_plus_13,RPM_Flag_plus_14,RPM_Flag_plus_15,RPM_Flag_plus_16:BOOL;

	RPM_Flag_minus_1,RPM_Flag_minus_2,RPM_Flag_minus_3,RPM_Flag_minus_4,RPM_Flag_minus_5,RPM_Flag_minus_6,RPM_Flag_minus_7,RPM_Flag_minus_8:BOOL;
	RPM_Flag_minus_9,RPM_Flag_minus_10,RPM_Flag_minus_11,RPM_Flag_minus_12,RPM_Flag_minus_13,RPM_Flag_minus_14,RPM_Flag_minus_15,RPM_Flag_minus_16:BOOL;

	RPM_Flag_CP_1,RPM_Flag_CP_2,RPM_Flag_CP_3,RPM_Flag_CP_4,RPM_Flag_CP_5,RPM_Flag_CP_6,RPM_Flag_CP_7,RPM_Flag_CP_8:BOOL;
	RPM_Flag_CP_9,RPM_Flag_CP_10,RPM_Flag_CP_11,RPM_Flag_CP_12,RPM_Flag_CP_13,RPM_Flag_CP_14,RPM_Flag_CP_15:BOOL;

	RPM_Flag_CN_2,RPM_Flag_CN_3,RPM_Flag_CN_4,RPM_Flag_CN_5,RPM_Flag_CN_6,RPM_Flag_CN_7,RPM_Flag_CN_8:BOOL;
	RPM_Flag_CN_9,RPM_Flag_CN_10,RPM_Flag_CN_11,RPM_Flag_CN_12,RPM_Flag_CN_13,RPM_Flag_CN_14,RPM_Flag_CN_15,RPM_Flag_CN_16:BOOL;

	(* для Turbo *)
	Turbo_Flag_plus_1,Turbo_Flag_plus_2,Turbo_Flag_plus_3,Turbo_Flag_plus_4,Turbo_Flag_plus_5,Turbo_Flag_plus_6,Turbo_Flag_plus_7,Turbo_Flag_plus_8:BOOL;
	Turbo_Flag_plus_9,Turbo_Flag_plus_10,Turbo_Flag_plus_11,Turbo_Flag_plus_12,Turbo_Flag_plus_13,Turbo_Flag_plus_14,Turbo_Flag_plus_15,Turbo_Flag_plus_16:BOOL;

	Turbo_Flag_minus_1,Turbo_Flag_minus_2,Turbo_Flag_minus_3,Turbo_Flag_minus_4,Turbo_Flag_minus_5,Turbo_Flag_minus_6,Turbo_Flag_minus_7,Turbo_Flag_minus_8:BOOL;
	Turbo_Flag_minus_9,Turbo_Flag_minus_10,Turbo_Flag_minus_11,Turbo_Flag_minus_12,Turbo_Flag_minus_13,Turbo_Flag_minus_14,Turbo_Flag_minus_15,Turbo_Flag_minus_16:BOOL;

	Turbo_Flag_CP_1,Turbo_Flag_CP_2,Turbo_Flag_CP_3,Turbo_Flag_CP_4,Turbo_Flag_CP_5,Turbo_Flag_CP_6,Turbo_Flag_CP_7,Turbo_Flag_CP_8:BOOL;
	Turbo_Flag_CP_9,Turbo_Flag_CP_10,Turbo_Flag_CP_11,Turbo_Flag_CP_12,Turbo_Flag_CP_13,Turbo_Flag_CP_14,Turbo_Flag_CP_15:BOOL;

	Turbo_Flag_CN_2,Turbo_Flag_CN_3,Turbo_Flag_CN_4,Turbo_Flag_CN_5,Turbo_Flag_CN_6,Turbo_Flag_CN_7,Turbo_Flag_CN_8:BOOL;
	Turbo_Flag_CN_9,Turbo_Flag_CN_10,Turbo_Flag_CN_11,Turbo_Flag_CN_12,Turbo_Flag_CN_13,Turbo_Flag_CN_14,Turbo_Flag_CN_15,Turbo_Flag_CN_16:BOOL;

(* Выбор типа калибровки и диапазона PPS *)
	PPS_number:BYTE;				(* Может принимать значение от 1 до 8 по числу диапазонов PPS *)
	(* Буферный массив с которым идет работа, а потом он копируется в калибровку *)
	Buffer: ARRAY [1..16,1..16] OF FLS;
	(* Буферный массив с которым идет работа, а потом он копируется в калибровку сразу для 2-х калибруемых величин газа и дизеля *)
	Buffer_GD: ARRAY [1..16,1..16] OF Cal_data;
	(* Переменные для циклов, для перебора значений *)
	i,j,k:BYTE;
	Change_volume:WORD:=5;
	Calculate_volume:REAL:=3;
	(* Работа с EEPROM *)
	s16_Return    	: INT;
	fb_EepWrite   	: FB_x_eep_write;
	fb_EepRead  	: FB_x_eep_read;

	Red_cal_DF, Write_cal_DF:BOOL;
END_VAR
(*********************** Работа с главной калибровочной таблицей ********************************************)

(* Сохраняем или читаем калибровку в/из EEPROM *)
EEPROM_read_write();
(* Считать требуемые данные из калибровочной таблицы в окно редактора *)
Buffer_read_write();
(* Считать требуемые данные из калибровочной таблицы в окно редактора для газа и дизелчя *)
Buffer_GD_rw();
(* Обработка данных в окне буфера: увеличить все, уменьшить все, залить значение и т.д *)
Edit_function();
(* Выбираем тип топлива для калибровки *)
Choose_gas_or_diesel();
(* Обработка раскидок по диагонали *)
Diagonal();

(***************************************** RPM ********************************************************)
(* Добавляем фиксированное значение к текущему значению в строке RPM *)
RPM_plus();
(* Вычитаем фиксированное значение к текущему значению в строке RPM *)
RPM_minus();
(* Копируем предидущую строку RPM в текущую *)
RPM_copy_prev();
(* Копируем следующую строку RPM в текущую *)
RPM_copy_next();

(********************************************TURBO*****************************************************)
(* Добавляем фиксированное значение к текущему значению в столбце Turbo *)
Turbo_plus();
(* Вычитаем фиксированное значение к текущему значению в столбце TURBO *)
Turbo_minus();
(* Копируем предидущий столбец Tubor в текущий *)
Turbo_copy_prev();
(* Копируем следущзий столбец Tubor в текущий *)
Turbo_copy_next();
END_PROGRAM
ACTION Buffer_GD_rw:
(* Считать требуемые данные из калибровочной таблицы в окно редактора *)
IF Red_cal_DF THEN
				FOR i:=1 TO 13 DO
					FOR j:=1 TO 13 DO
							Buffer_GD[i,j].Gas:=p.Cal_table[i,j].GAS;
							Buffer_GD[i,j].Diesel:=p.Cal_table[i,j].Diesel;
					END_FOR
				END_FOR
	Red_cal_DF:=FALSE;
END_IF

(* Записать текущие данные из окна редактора в калибровочную таблицу *)
IF Write_cal_DF THEN

				FOR i:=1 TO 13 DO
					FOR j:=1 TO 13 DO
							p.Cal_table[i,j].GAS:=WORD_TO_BYTE(Buffer_GD[i,j].Gas);
							p.Cal_table[i,j].Diesel:=WORD_TO_BYTE(Buffer_GD[i,j].Diesel);
					END_FOR
				END_FOR

	Write_cal_DF:=FALSE;
END_IF
END_ACTION
ACTION Buffer_read_write:
(* Считать требуемые данные из калибровочной таблицы в окно редактора *)
IF Red_cal2 THEN

				FOR i:=1 TO 16 DO
					FOR j:=1 TO 16 DO
					(* Работа или с газовой или с дизельной калибровкой *)
						IF Flag_cal_table_gas THEN
							Buffer[i,j].a:=p.Cal_table[i,j].GAS;
						ELSE
							Buffer[i,j].a:=p.Cal_table[i,j].Diesel;
						END_IF
					END_FOR
				END_FOR

	Red_cal2:=FALSE;
END_IF

(* Записать текущие данные из окна редактора в калибровочную таблицу *)
IF Write_cal2 THEN

				FOR i:=1 TO 16 DO
					FOR j:=1 TO 16 DO
						(* Работа или с газовой или с дизельной калибровкой *)
						IF Flag_cal_table_gas THEN
							p.Cal_table[i,j].GAS:=WORD_TO_BYTE(Buffer[i,j].a);
						ELSE
							p.Cal_table[i,j].Diesel:=WORD_TO_BYTE(Buffer[i,j].a);
						END_IF;
					END_FOR
				END_FOR

	Write_cal2:=FALSE;
END_IF
END_ACTION
ACTION Choose_gas_or_diesel:
(* Выбираем тип топлива для калибровки *)

IF Flag_cal_table_gas THEN
	Fuel_type:='GAS';
ELSE
	Fuel_type:='DIESEL';
END_IF
END_ACTION
ACTION Diagonal:
(**************************************** ДИАГОНАЛЬНЫЕ КАЛИБРОВКИ ***********************************************)

(* Устанавливаем симметричную диагональную калибровку с шагом 1 в окне редактора *)
IF Diagonal_1 THEN
				i:=17;
				WHILE i<>0  DO
						i:=i-1;
						j:=17;
						WHILE j<>0 DO
						j:=j-1;
							IF j=16 AND i=16 THEN
								Buffer[i,j].a:=Change_volume;
							ELSIF j=16 THEN
								(* Почему то если получается отрицательное значение в массиве, возникает ошибка, для предотвращения проверяем это явно *)
								IF Buffer[i+1,j].a >= 1 THEN
									Buffer[i,j].a:=Buffer[i+1,j].a-1;
								ELSE
									Buffer[i,j].a:=0;
								END_IF
							ELSE
								IF Buffer[i,j+1].a >= 1 THEN
									Buffer[i,j].a:=Buffer[i,j+1].a-1;
								ELSE
									Buffer[i,j].a:=0;
								END_IF
							END_IF
						END_WHILE
				END_WHILE
				Diagonal_1:=FALSE;
END_IF

(* Устанавливаем симметричную диагональную калибровку с шагом 2 в окне редактора *)
IF Diagonal_2 THEN
				i:=17;
				WHILE i<>0  DO
						i:=i-1;
						j:=17;
						WHILE j<>0 DO
						j:=j-1;
							IF j=16 AND i=16 THEN
								Buffer[i,j].a:=Change_volume;
							ELSIF j=16 THEN
								(* Почему то если получается отрицательное значение в массиве, возникает ошибка, для предотвращения проверяем это явно *)
								IF Buffer[i+1,j].a >= 2 THEN
									Buffer[i,j].a:=Buffer[i+1,j].a-2;
								ELSE
									Buffer[i,j].a:=0;
								END_IF
							ELSE
								IF Buffer[i,j+1].a >= 2 THEN
									Buffer[i,j].a:=Buffer[i,j+1].a-2;
								ELSE
									Buffer[i,j].a:=0;
								END_IF
							END_IF
						END_WHILE
				END_WHILE
				Diagonal_2:=FALSE;
END_IF

(* Устанавливаем симметричную диагональную калибровку с шагом 3 в окне редактора *)
IF Diagonal_3 THEN
				i:=17;
				WHILE i<>0  DO
						i:=i-1;
						j:=17;
						WHILE j<>0 DO
						j:=j-1;
							IF j=16 AND i=16 THEN
								Buffer[i,j].a:=Change_volume;
							ELSIF j=16 THEN
								(* Почему то если получается отрицательное значение в массиве, возникает ошибка, для предотвращения проверяем это явно *)
								IF Buffer[i+1,j].a >= 3 THEN
									Buffer[i,j].a:=Buffer[i+1,j].a-3;
								ELSE
									Buffer[i,j].a:=0;
								END_IF
							ELSE
								IF Buffer[i,j+1].a >= 3 THEN
									Buffer[i,j].a:=Buffer[i,j+1].a-3;
								ELSE
									Buffer[i,j].a:=0;
								END_IF
							END_IF
						END_WHILE
				END_WHILE
				Diagonal_3:=FALSE;
END_IF

(* Устанавливаем симметричную диагональную калибровку с шагом 2 по горизонтали  и 1 по вертикале в окне редактора *)
IF Diagonal_21 THEN
				i:=17;
				WHILE i<>0  DO
						i:=i-1;
						j:=17;
						WHILE j<>0 DO
						j:=j-1;
							IF j=16 AND i=16 THEN
								Buffer[i,j].a:=Change_volume;
							ELSIF j=16 THEN
								(* Почему то если получается отрицательное значение в массиве, возникает ошибка, для предотвращения проверяем это явно *)
								IF Buffer[i+1,j].a >= 2 THEN
									Buffer[i,j].a:=Buffer[i+1,j].a-2;
								ELSE
									Buffer[i,j].a:=0;
								END_IF
							ELSE
								IF Buffer[i,j+1].a >= 1 THEN
									Buffer[i,j].a:=Buffer[i,j+1].a-1;
								ELSE
									Buffer[i,j].a:=0;
								END_IF
							END_IF
						END_WHILE
				END_WHILE
				Diagonal_21:=FALSE;
END_IF
(* Устанавливаем симметричную диагональную калибровку с шагом 3 по горизонтали  и 1 по вертикале в окне редактора *)
IF Diagonal_31 THEN
				i:=17;
				WHILE i<>0  DO
						i:=i-1;
						j:=17;
						WHILE j<>0 DO
						j:=j-1;
							IF j=16 AND i=16 THEN
								Buffer[i,j].a:=Change_volume;
							ELSIF j=16 THEN
								(* Почему то если получается отрицательное значение в массиве, возникает ошибка, для предотвращения проверяем это явно *)
								IF Buffer[i+1,j].a >= 3 THEN
									Buffer[i,j].a:=Buffer[i+1,j].a-3;
								ELSE
									Buffer[i,j].a:=0;
								END_IF
							ELSE
								IF Buffer[i,j+1].a >= 1 THEN
									Buffer[i,j].a:=Buffer[i,j+1].a-1;
								ELSE
									Buffer[i,j].a:=0;
								END_IF
							END_IF
						END_WHILE
				END_WHILE
				Diagonal_31:=FALSE;
END_IF

(* Устанавливаем симметричную диагональную калибровку с шагом 3 по горизонтали  и 2 по вертикале в окне редактора *)
IF Diagonal_32 THEN
				i:=17;
				WHILE i<>0  DO
						i:=i-1;
						j:=17;
						WHILE j<>0 DO
						j:=j-1;
							IF j=16 AND i=16 THEN
								Buffer[i,j].a:=Change_volume;
							ELSIF j=16 THEN
								(* Почему то если получается отрицательное значение в массиве, возникает ошибка, для предотвращения проверяем это явно *)
								IF Buffer[i+1,j].a >= 3 THEN
									Buffer[i,j].a:=Buffer[i+1,j].a-3;
								ELSE
									Buffer[i,j].a:=0;
								END_IF
							ELSE
								IF Buffer[i,j+1].a >= 2 THEN
									Buffer[i,j].a:=Buffer[i,j+1].a-2;
								ELSE
									Buffer[i,j].a:=0;
								END_IF
							END_IF
						END_WHILE
				END_WHILE
				Diagonal_32:=FALSE;
END_IF
END_ACTION
ACTION Edit_function:
(********************************* Функции редактирования ***********************************************)

IF Flag_cal_table_gas = FALSE THEN
	(* Работа с дизельной калибровкой *)
	(* Автоматически расчитать эмуляцию от подачи газа *)
	IF Calculate THEN
			FOR i:=1 TO 16 DO
				FOR j:=1 TO 16 DO
						p.Cal_table[i,j].DIESEL:= REAL_TO_BYTE(p.Cal_table[i,j].GAS*Calculate_volume);
						Buffer[i,j].a:=p.Cal_table[i,j].DIESEL;
				END_FOR
			END_FOR
		Calculate:=FALSE;
	END_IF
END_IF

(************ Работа с буффером ***********************************)

(* Устанавливаем в определенное значение все значения в окне редактора *)
IF Set_ALL THEN
				FOR i:=1 TO 16 DO
						FOR j:=1 TO 16 DO
							Buffer[i,j].a:=Change_volume;
						END_FOR
				END_FOR
				Set_ALL:=FALSE;
END_IF

(* Устанавливаем в определенное значение нижнюю диагональ  в окне редактора *)
IF HALF_set_ALL THEN
				k:=17;
				i:=17;
				FOR j:=1 TO 16 DO
					k:=k-1;
					i:=17;
						WHILE i<>k  DO
							i:=i-1;
							Buffer[i,j].a:=Change_volume;
						END_WHILE
				END_FOR
				HALF_set_ALL:=FALSE;
END_IF

(* Увеличиваем все значения  в окне редактора *)
IF ALL_plus THEN
				FOR i:=1 TO 16 DO
						FOR j:=1 TO 16 DO
									Buffer[i,j].a:=Buffer[i,j].a+Change_volume;
						END_FOR
				END_FOR
				ALL_plus:=FALSE;
END_IF

(* Уменьшаем все значения  в окне редактора *)
IF ALL_minus THEN
				FOR i:=1 TO 16 DO
						FOR j:=1 TO 16 DO
							Buffer[i,j].a:=Buffer[i,j].a-Change_volume;
							(* Если из за уменьшения значения перешли 0 и стали слишком большими сбросить в 0 *)
							IF Buffer[i,j].a > 200 THEN
								Buffer[i,j].a:=0;
							END_IF
						END_FOR
				END_FOR
				ALL_minus:=FALSE;
END_IF
END_ACTION
ACTION EEPROM_read_write:
(* Сохраняем калибровку в файле *)
IF Write_Cal THEN
	fb_EepWrite(ou32_Address:=0, ou32_Count:=SIZEOF(p), opu8_Data:=ADR(p), os16_Status=>s16_Return);
	Write_cal:=FALSE;
END_IF

(* Читаем калибровку из файла *)
IF Read_Cal THEN
	fb_EepRead(ou32_Address:=0, ou32_Count:=SIZEOF(p), opu8_Data:=ADR(p), os16_Status=>s16_Return);
	Read_cal:=FALSE;
END_IF
END_ACTION
ACTION RPM_copy_next:
(* Копируем следующую строку RPM в текущую *)
IF RPM_Flag_CP_1 THEN
	FOR i:=1 TO 16 DO
		Buffer[i,1].a:=Buffer[i,2].a;
	END_FOR
	RPM_Flag_CP_1:=FALSE;
END_IF
IF RPM_Flag_CP_2 THEN
	FOR i:=1 TO 16 DO
		Buffer[i,2].a:=Buffer[i,3].a;
	END_FOR
	RPM_Flag_CP_2:=FALSE;
END_IF
IF RPM_Flag_CP_3 THEN
	FOR i:=1 TO 16 DO
		Buffer[i,3].a:=Buffer[i,4].a;
	END_FOR
	RPM_Flag_CP_3:=FALSE;
END_IF
IF RPM_Flag_CP_4 THEN
	FOR i:=1 TO 16 DO
		Buffer[i,4].a:=Buffer[i,5].a;
	END_FOR
	RPM_Flag_CP_4:=FALSE;
END_IF
IF RPM_Flag_CP_5 THEN
	FOR i:=1 TO 16 DO
		Buffer[i,5].a:=Buffer[i,6].a;
	END_FOR
	RPM_Flag_CP_5:=FALSE;
END_IF
IF RPM_Flag_CP_6 THEN
	FOR i:=1 TO 16 DO
		Buffer[i,6].a:=Buffer[i,7].a;
	END_FOR
	RPM_Flag_CP_6:=FALSE;
END_IF
IF RPM_Flag_CP_7 THEN
	FOR i:=1 TO 16 DO
		Buffer[i,7].a:=Buffer[i,8].a;
	END_FOR
	RPM_Flag_CP_7:=FALSE;
END_IF
IF RPM_Flag_CP_8 THEN
	FOR i:=1 TO 16 DO
		Buffer[i,8].a:=Buffer[i,9].a;
	END_FOR
	RPM_Flag_CP_8:=FALSE;
END_IF

IF RPM_Flag_CP_9 THEN
	FOR i:=1 TO 16 DO
		Buffer[i,9].a:=Buffer[i,10].a;
	END_FOR
	RPM_Flag_CP_9:=FALSE;
END_IF
IF RPM_Flag_CP_10 THEN
	FOR i:=1 TO 16 DO
		Buffer[i,10].a:=Buffer[i,11].a;
	END_FOR
	RPM_Flag_CP_10:=FALSE;
END_IF
IF RPM_Flag_CP_11 THEN
	FOR i:=1 TO 16 DO
		Buffer[i,11].a:=Buffer[i,12].a;
	END_FOR
	RPM_Flag_CP_11:=FALSE;
END_IF
IF RPM_Flag_CP_12 THEN
	FOR i:=1 TO 16 DO
		Buffer[i,12].a:=Buffer[i,13].a;
	END_FOR
	RPM_Flag_CP_12:=FALSE;
END_IF
IF RPM_Flag_CP_13 THEN
	FOR i:=1 TO 16 DO
		Buffer[i,13].a:=Buffer[i,14].a;
	END_FOR
	RPM_Flag_CP_13:=FALSE;
END_IF
IF RPM_Flag_CP_14 THEN
	FOR i:=1 TO 16 DO
		Buffer[i,14].a:=Buffer[i,15].a;
	END_FOR
	RPM_Flag_CP_14:=FALSE;
END_IF
IF RPM_Flag_CP_15 THEN
	FOR i:=1 TO 16 DO
		Buffer[i,15].a:=Buffer[i,16].a;
	END_FOR
	RPM_Flag_CP_15:=FALSE;
END_IF
END_ACTION
ACTION RPM_copy_prev:
(* Копируем предидущую строку RPM в текущую *)

IF RPM_Flag_CN_2 THEN
	FOR i:=1 TO 16 DO
		Buffer[i,2].a:=Buffer[i,1].a;
	END_FOR
	RPM_Flag_CN_2:=FALSE;
END_IF
IF RPM_Flag_CN_3 THEN
	FOR i:=1 TO 16 DO
		Buffer[i,3].a:=Buffer[i,2].a;
	END_FOR
	RPM_Flag_CN_3:=FALSE;
END_IF
IF RPM_Flag_CN_4 THEN
	FOR i:=1 TO 16 DO
		Buffer[i,4].a:=Buffer[i,3].a;
	END_FOR
	RPM_Flag_CN_4:=FALSE;
END_IF
IF RPM_Flag_CN_5 THEN
	FOR i:=1 TO 16 DO
		Buffer[i,5].a:=Buffer[i,4].a;
	END_FOR
	RPM_Flag_CN_5:=FALSE;
END_IF
IF RPM_Flag_CN_6 THEN
	FOR i:=1 TO 16 DO
		Buffer[i,6].a:=Buffer[i,5].a;
	END_FOR
	RPM_Flag_CN_6:=FALSE;
END_IF
IF RPM_Flag_CN_7 THEN
	FOR i:=1 TO 16 DO
		Buffer[i,7].a:=Buffer[i,6].a;
	END_FOR
	RPM_Flag_CN_7:=FALSE;
END_IF
IF RPM_Flag_CN_8 THEN
	FOR i:=1 TO 16 DO
		Buffer[i,8].a:=Buffer[i,7].a;
	END_FOR
	RPM_Flag_CN_8:=FALSE;
END_IF

IF RPM_Flag_CN_9 THEN
	FOR i:=1 TO 16 DO
		Buffer[i,9].a:=Buffer[i,8].a;
	END_FOR
	RPM_Flag_CN_9:=FALSE;
END_IF
IF RPM_Flag_CN_10 THEN
	FOR i:=1 TO 16 DO
		Buffer[i,10].a:=Buffer[i,9].a;
	END_FOR
	RPM_Flag_CN_10:=FALSE;
END_IF
IF RPM_Flag_CN_11 THEN
	FOR i:=1 TO 16 DO
		Buffer[i,11].a:=Buffer[i,10].a;
	END_FOR
	RPM_Flag_CN_11:=FALSE;
END_IF
IF RPM_Flag_CN_12 THEN
	FOR i:=1 TO 16 DO
		Buffer[i,12].a:=Buffer[i,11].a;
	END_FOR
	RPM_Flag_CN_12:=FALSE;
END_IF
IF RPM_Flag_CN_13 THEN
	FOR i:=1 TO 16 DO
		Buffer[i,13].a:=Buffer[i,12].a;
	END_FOR
	RPM_Flag_CN_13:=FALSE;
END_IF
IF RPM_Flag_CN_14 THEN
	FOR i:=1 TO 16 DO
		Buffer[i,14].a:=Buffer[i,13].a;
	END_FOR
	RPM_Flag_CN_14:=FALSE;
END_IF
IF RPM_Flag_CN_15 THEN
	FOR i:=1 TO 16 DO
		Buffer[i,15].a:=Buffer[i,14].a;
	END_FOR
	RPM_Flag_CN_15:=FALSE;
END_IF
IF RPM_Flag_CN_16 THEN
	FOR i:=1 TO 16 DO
		Buffer[i,16].a:=Buffer[i,15].a;
	END_FOR
	RPM_Flag_CN_16:=FALSE;
END_IF
END_ACTION
ACTION RPM_minus:
(* Вычитаем фиксированное значение к текущему значению в строке RPM *)

IF RPM_Flag_minus_1 THEN
	FOR i:=1 TO 16 DO
		Buffer[i,1].a:=Buffer[i,1].a-Change_volume;
		(* Если из за уменьшения значения перешли 0 и стали слишком большими сбросить в 0 *)
		IF Buffer[i,1].a > 200 THEN
			Buffer[i,1].a:=0;
		END_IF
	END_FOR
	RPM_Flag_minus_1:=FALSE;
END_IF
IF RPM_Flag_minus_2 THEN
	FOR i:=1 TO 16 DO
		Buffer[i,2].a:=Buffer[i,2].a-Change_volume;
		(* Если из за уменьшения значения перешли 0 и стали слишком большими сбросить в 0 *)
		IF Buffer[i,2].a > 200 THEN
			Buffer[i,2].a:=0;
		END_IF
	END_FOR
	RPM_Flag_minus_2:=FALSE;
END_IF
IF RPM_Flag_minus_3 THEN
	FOR i:=1 TO 16 DO
		Buffer[i,3].a:=Buffer[i,3].a-Change_volume;
		(* Если из за уменьшения значения перешли 0 и стали слишком большими сбросить в 0 *)
		IF Buffer[i,3].a > 200 THEN
			Buffer[i,3].a:=0;
		END_IF
	END_FOR
	RPM_Flag_minus_3:=FALSE;
END_IF
IF RPM_Flag_minus_4 THEN
	FOR i:=1 TO 16 DO
		Buffer[i,4].a:=Buffer[i,4].a-Change_volume;
		(* Если из за уменьшения значения перешли 0 и стали слишком большими сбросить в 0 *)
		IF Buffer[i,4].a > 200 THEN
			Buffer[i,4].a:=0;
		END_IF
	END_FOR
	RPM_Flag_minus_4:=FALSE;
END_IF
IF RPM_Flag_minus_5 THEN
	FOR i:=1 TO 16 DO
		Buffer[i,5].a:=Buffer[i,5].a-Change_volume;
		(* Если из за уменьшения значения перешли 0 и стали слишком большими сбросить в 0 *)
		IF Buffer[i,5].a > 200 THEN
			Buffer[i,5].a:=0;
		END_IF
	END_FOR
	RPM_Flag_minus_5:=FALSE;
END_IF
IF RPM_Flag_minus_6 THEN
	FOR i:=1 TO 16 DO
		Buffer[i,6].a:=Buffer[i,6].a-Change_volume;
		(* Если из за уменьшения значения перешли 0 и стали слишком большими сбросить в 0 *)
		IF Buffer[i,6].a > 200 THEN
			Buffer[i,6].a:=0;
		END_IF
	END_FOR
	RPM_Flag_minus_6:=FALSE;
END_IF
IF RPM_Flag_minus_7 THEN
	FOR i:=1 TO 16 DO
		Buffer[i,7].a:=Buffer[i,7].a-Change_volume;
		(* Если из за уменьшения значения перешли 0 и стали слишком большими сбросить в 0 *)
		IF Buffer[i,7].a > 200 THEN
			Buffer[i,7].a:=0;
		END_IF
	END_FOR
	RPM_Flag_minus_7:=FALSE;
END_IF
IF RPM_Flag_minus_8 THEN
	FOR i:=1 TO 16 DO
		Buffer[i,8].a:=Buffer[i,8].a-Change_volume;
		(* Если из за уменьшения значения перешли 0 и стали слишком большими сбросить в 0 *)
		IF Buffer[i,8].a > 200 THEN
			Buffer[i,8].a:=0;
		END_IF
	END_FOR
	RPM_Flag_minus_8:=FALSE;
END_IF

IF RPM_Flag_minus_9 THEN
	FOR i:=1 TO 16 DO
		Buffer[i,9].a:=Buffer[i,9].a-Change_volume;
		(* Если из за уменьшения значения перешли 0 и стали слишком большими сбросить в 0 *)
		IF Buffer[i,9].a > 100 THEN
			Buffer[i,9].a:=0;
		END_IF
	END_FOR
	RPM_Flag_minus_9:=FALSE;
END_IF
IF RPM_Flag_minus_10 THEN
	FOR i:=1 TO 16 DO
		Buffer[i,10].a:=Buffer[i,10].a-Change_volume;
		(* Если из за уменьшения значения перешли 0 и стали слишком большими сбросить в 0 *)
		IF Buffer[i,10].a > 200 THEN
			Buffer[i,10].a:=0;
		END_IF
	END_FOR
	RPM_Flag_minus_10:=FALSE;
END_IF
IF RPM_Flag_minus_11 THEN
	FOR i:=1 TO 16 DO
		Buffer[i,11].a:=Buffer[i,11].a-Change_volume;
		(* Если из за уменьшения значения перешли 0 и стали слишком большими сбросить в 0 *)
		IF Buffer[i,11].a > 200 THEN
			Buffer[i,11].a:=0;
		END_IF
	END_FOR
	RPM_Flag_minus_11:=FALSE;
END_IF
IF RPM_Flag_minus_12 THEN
	FOR i:=1 TO 16 DO
		Buffer[i,12].a:=Buffer[i,12].a-Change_volume;
		(* Если из за уменьшения значения перешли 0 и стали слишком большими сбросить в 0 *)
		IF Buffer[i,12].a > 200 THEN
			Buffer[i,12].a:=0;
		END_IF
	END_FOR
	RPM_Flag_minus_12:=FALSE;
END_IF
IF RPM_Flag_minus_13 THEN
	FOR i:=1 TO 16 DO
		Buffer[i,13].a:=Buffer[i,13].a-Change_volume;
		(* Если из за уменьшения значения перешли 0 и стали слишком большими сбросить в 0 *)
		IF Buffer[i,13].a > 200 THEN
			Buffer[i,13].a:=0;
		END_IF
	END_FOR
	RPM_Flag_minus_13:=FALSE;
END_IF
IF RPM_Flag_minus_14 THEN
	FOR i:=1 TO 16 DO
		Buffer[i,14].a:=Buffer[i,14].a-Change_volume;
		(* Если из за уменьшения значения перешли 0 и стали слишком большими сбросить в 0 *)
		IF Buffer[i,14].a > 200 THEN
			Buffer[i,14].a:=0;
		END_IF
	END_FOR
	RPM_Flag_minus_14:=FALSE;
END_IF
IF RPM_Flag_minus_15 THEN
	FOR i:=1 TO 16 DO
		Buffer[i,15].a:=Buffer[i,15].a-Change_volume;
		(* Если из за уменьшения значения перешли 0 и стали слишком большими сбросить в 0 *)
		IF Buffer[i,15].a > 200 THEN
			Buffer[i,15].a:=0;
		END_IF
	END_FOR
	RPM_Flag_minus_15:=FALSE;
END_IF
IF RPM_Flag_minus_16 THEN
	FOR i:=1 TO 16 DO
		Buffer[i,16].a:=Buffer[i,16].a-Change_volume;
		(* Если из за уменьшения значения перешли 0 и стали слишком большими сбросить в 0 *)
		IF Buffer[i,16].a > 200 THEN
			Buffer[i,16].a:=0;
		END_IF
	END_FOR
	RPM_Flag_minus_16:=FALSE;
END_IF
END_ACTION
ACTION RPM_plus:
(* Добавляем фиксированное значение к текущему значению в строке RPM *)

IF RPM_Flag_plus_1 THEN
	FOR i:=1 TO 16 DO
		Buffer[i,1].a:=Buffer[i,1].a+Change_volume;
	END_FOR
	RPM_Flag_plus_1:=FALSE;
END_IF
IF RPM_Flag_plus_2 THEN
	FOR i:=1 TO 16 DO
		Buffer[i,2].a:=Buffer[i,2].a+Change_volume;
	END_FOR
	RPM_Flag_plus_2:=FALSE;
END_IF
IF RPM_Flag_plus_3 THEN
	FOR i:=1 TO 16 DO
		Buffer[i,3].a:=Buffer[i,3].a+Change_volume;
	END_FOR
	RPM_Flag_plus_3:=FALSE;
END_IF
IF RPM_Flag_plus_4 THEN
	FOR i:=1 TO 16 DO
		Buffer[i,4].a:=Buffer[i,4].a+Change_volume;
	END_FOR
	RPM_Flag_plus_4:=FALSE;
END_IF
IF RPM_Flag_plus_5 THEN
	FOR i:=1 TO 16 DO
		Buffer[i,5].a:=Buffer[i,5].a+Change_volume;
	END_FOR
	RPM_Flag_plus_5:=FALSE;
END_IF
IF RPM_Flag_plus_6 THEN
	FOR i:=1 TO 16 DO
		Buffer[i,6].a:=Buffer[i,6].a+Change_volume;
	END_FOR
	RPM_Flag_plus_6:=FALSE;
END_IF
IF RPM_Flag_plus_7 THEN
	FOR i:=1 TO 16 DO
		Buffer[i,7].a:=Buffer[i,7].a+Change_volume;
	END_FOR
	RPM_Flag_plus_7:=FALSE;
END_IF
IF RPM_Flag_plus_8 THEN
	FOR i:=1 TO 16 DO
		Buffer[i,8].a:=Buffer[i,8].a+Change_volume;
	END_FOR
	RPM_Flag_plus_8:=FALSE;
END_IF


IF RPM_Flag_plus_9 THEN
	FOR i:=1 TO 16 DO
		Buffer[i,9].a:=Buffer[i,9].a+Change_volume;
	END_FOR
	RPM_Flag_plus_9:=FALSE;
END_IF
IF RPM_Flag_plus_10 THEN
	FOR i:=1 TO 16 DO
		Buffer[i,10].a:=Buffer[i,10].a+Change_volume;
	END_FOR
	RPM_Flag_plus_10:=FALSE;
END_IF
IF RPM_Flag_plus_11 THEN
	FOR i:=1 TO 16 DO
		Buffer[i,11].a:=Buffer[i,11].a+Change_volume;
	END_FOR
	RPM_Flag_plus_11:=FALSE;
END_IF
IF RPM_Flag_plus_12 THEN
	FOR i:=1 TO 16 DO
		Buffer[i,12].a:=Buffer[i,12].a+Change_volume;
	END_FOR
	RPM_Flag_plus_12:=FALSE;
END_IF
IF RPM_Flag_plus_13 THEN
	FOR i:=1 TO 16 DO
		Buffer[i,13].a:=Buffer[i,13].a+Change_volume;
	END_FOR
	RPM_Flag_plus_13:=FALSE;
END_IF
IF RPM_Flag_plus_14 THEN
	FOR i:=1 TO 16 DO
		Buffer[i,14].a:=Buffer[i,14].a+Change_volume;
	END_FOR
	RPM_Flag_plus_14:=FALSE;
END_IF
IF RPM_Flag_plus_15 THEN
	FOR i:=1 TO 16 DO
		Buffer[i,15].a:=Buffer[i,15].a+Change_volume;
	END_FOR
	RPM_Flag_plus_15:=FALSE;
END_IF
IF RPM_Flag_plus_16 THEN
	FOR i:=1 TO 16 DO
		Buffer[i,16].a:=Buffer[i,16].a+Change_volume;
	END_FOR
	RPM_Flag_plus_16:=FALSE;
END_IF
END_ACTION
ACTION Turbo_copy_next:
(* Копируем следующий столбец Turbo в текущий *)
IF Turbo_Flag_CP_1 THEN
	FOR i:=1 TO 16 DO
		Buffer[1,i].a:=Buffer[2,i].a;
	END_FOR
	Turbo_Flag_CP_1:=FALSE;
END_IF
IF Turbo_Flag_CP_2 THEN
	FOR i:=1 TO 16 DO
		Buffer[2,i].a:=Buffer[3,i].a;
	END_FOR
	Turbo_Flag_CP_2:=FALSE;
END_IF
IF Turbo_Flag_CP_3 THEN
	FOR i:=1 TO 16 DO
		Buffer[3,i].a:=Buffer[4,i].a;
	END_FOR
	Turbo_Flag_CP_3:=FALSE;
END_IF
IF Turbo_Flag_CP_4 THEN
	FOR i:=1 TO 16 DO
		Buffer[4,i].a:=Buffer[5,i].a;
	END_FOR
	Turbo_Flag_CP_4:=FALSE;
END_IF
IF Turbo_Flag_CP_5 THEN
	FOR i:=1 TO 16 DO
		Buffer[5,i].a:=Buffer[6,i].a;
	END_FOR
	Turbo_Flag_CP_5:=FALSE;
END_IF
IF Turbo_Flag_CP_6 THEN
	FOR i:=1 TO 16 DO
		Buffer[6,i].a:=Buffer[7,i].a;
	END_FOR
	Turbo_Flag_CP_6:=FALSE;
END_IF
IF Turbo_Flag_CP_7 THEN
	FOR i:=1 TO 16 DO
		Buffer[7,i].a:=Buffer[8,i].a;
	END_FOR
	Turbo_Flag_CP_7:=FALSE;
END_IF
IF Turbo_Flag_CP_8 THEN
	FOR i:=1 TO 16 DO
		Buffer[8,i].a:=Buffer[9,i].a;
	END_FOR
	Turbo_Flag_CP_8:=FALSE;
END_IF

IF Turbo_Flag_CP_9 THEN
	FOR i:=1 TO 16 DO
		Buffer[9,i].a:=Buffer[10,i].a;
	END_FOR
	Turbo_Flag_CP_9:=FALSE;
END_IF
IF Turbo_Flag_CP_10 THEN
	FOR i:=1 TO 16 DO
		Buffer[10,i].a:=Buffer[11,i].a;
	END_FOR
	Turbo_Flag_CP_10:=FALSE;
END_IF
IF Turbo_Flag_CP_11 THEN
	FOR i:=1 TO 16 DO
		Buffer[11,i].a:=Buffer[12,i].a;
	END_FOR
	Turbo_Flag_CP_11:=FALSE;
END_IF
IF Turbo_Flag_CP_12 THEN
	FOR i:=1 TO 16 DO
		Buffer[12,i].a:=Buffer[13,i].a;
	END_FOR
	Turbo_Flag_CP_12:=FALSE;
END_IF
IF Turbo_Flag_CP_13 THEN
	FOR i:=1 TO 16 DO
		Buffer[13,i].a:=Buffer[14,i].a;
	END_FOR
	Turbo_Flag_CP_13:=FALSE;
END_IF
IF Turbo_Flag_CP_14 THEN
	FOR i:=1 TO 16 DO
		Buffer[14,i].a:=Buffer[15,i].a;
	END_FOR
	Turbo_Flag_CP_14:=FALSE;
END_IF
IF Turbo_Flag_CP_15 THEN
	FOR i:=1 TO 16 DO
		Buffer[15,i].a:=Buffer[16,i].a;
	END_FOR
	Turbo_Flag_CP_15:=FALSE;
END_IF
END_ACTION
ACTION Turbo_copy_prev:
(* Копируем предидущий столбец Turbo в текущий *)

IF Turbo_Flag_CN_2 THEN
	FOR i:=1 TO 16 DO
		Buffer[2,i].a:=Buffer[1,i].a;
	END_FOR
	Turbo_Flag_CN_2:=FALSE;
END_IF
IF Turbo_Flag_CN_3 THEN
	FOR i:=1 TO 16 DO
		Buffer[3,i].a:=Buffer[2,i].a;
	END_FOR
	Turbo_Flag_CN_3:=FALSE;
END_IF
IF Turbo_Flag_CN_4 THEN
	FOR i:=1 TO 16 DO
		Buffer[4,i].a:=Buffer[3,i].a;
	END_FOR
	Turbo_Flag_CN_4:=FALSE;
END_IF
IF Turbo_Flag_CN_5 THEN
	FOR i:=1 TO 16 DO
		Buffer[5,i].a:=Buffer[4,i].a;
	END_FOR
	Turbo_Flag_CN_5:=FALSE;
END_IF
IF Turbo_Flag_CN_6 THEN
	FOR i:=1 TO 16 DO
		Buffer[6,i].a:=Buffer[5,i].a;
	END_FOR
	Turbo_Flag_CN_6:=FALSE;
END_IF
IF Turbo_Flag_CN_7 THEN
	FOR i:=1 TO 16 DO
		Buffer[7,i].a:=Buffer[6,i].a;
	END_FOR
	Turbo_Flag_CN_7:=FALSE;
END_IF
IF Turbo_Flag_CN_8 THEN
	FOR i:=1 TO 16 DO
		Buffer[8,i].a:=Buffer[7,i].a;
	END_FOR
	Turbo_Flag_CN_8:=FALSE;
END_IF

IF Turbo_Flag_CN_9 THEN
	FOR i:=1 TO 16 DO
		Buffer[9,i].a:=Buffer[8,i].a;
	END_FOR
	Turbo_Flag_CN_9:=FALSE;
END_IF
IF Turbo_Flag_CN_10 THEN
	FOR i:=1 TO 16 DO
		Buffer[10,i].a:=Buffer[9,i].a;
	END_FOR
	Turbo_Flag_CN_10:=FALSE;
END_IF
IF Turbo_Flag_CN_11 THEN
	FOR i:=1 TO 16 DO
		Buffer[11,i].a:=Buffer[10,i].a;
	END_FOR
	Turbo_Flag_CN_11:=FALSE;
END_IF
IF Turbo_Flag_CN_12 THEN
	FOR i:=1 TO 16 DO
		Buffer[12,i].a:=Buffer[11,i].a;
	END_FOR
	Turbo_Flag_CN_12:=FALSE;
END_IF
IF Turbo_Flag_CN_13 THEN
	FOR i:=1 TO 16 DO
		Buffer[13,i].a:=Buffer[12,i].a;
	END_FOR
	Turbo_Flag_CN_13:=FALSE;
END_IF
IF Turbo_Flag_CN_14 THEN
	FOR i:=1 TO 16 DO
		Buffer[14,i].a:=Buffer[13,i].a;
	END_FOR
	Turbo_Flag_CN_14:=FALSE;
END_IF
IF Turbo_Flag_CN_15 THEN
	FOR i:=1 TO 16 DO
		Buffer[15,i].a:=Buffer[14,i].a;
	END_FOR
	Turbo_Flag_CN_15:=FALSE;
END_IF
IF Turbo_Flag_CN_16 THEN
	FOR i:=1 TO 16 DO
		Buffer[16,i].a:=Buffer[15,i].a;
	END_FOR
	Turbo_Flag_CN_16:=FALSE;
END_IF
END_ACTION
ACTION Turbo_minus:
(* Вычитаем фиксированное значение к текущему значению в столбце TURBO *)

IF Turbo_Flag_minus_1 THEN
	FOR i:=1 TO 16 DO
		Buffer[1,i].a:=Buffer[1,i].a-Change_volume;
		(* Если из за уменьшения значения перешли 0 и стали слишком большими сбросить в 0 *)
		IF Buffer[1,i].a > 200 THEN
			Buffer[1,i].a:=0;
		END_IF
	END_FOR
	Turbo_Flag_minus_1:=FALSE;
END_IF
IF Turbo_Flag_minus_2 THEN
	FOR i:=1 TO 16 DO
		Buffer[2,i].a:=Buffer[2,i].a-Change_volume;
		(* Если из за уменьшения значения перешли 0 и стали слишком большими сбросить в 0 *)
		IF Buffer[2,i].a > 200 THEN
			Buffer[2,i].a:=0;
		END_IF
	END_FOR
	Turbo_Flag_minus_2:=FALSE;
END_IF
IF Turbo_Flag_minus_3 THEN
	FOR i:=1 TO 16 DO
		Buffer[3,i].a:=Buffer[3,i].a-Change_volume;
		(* Если из за уменьшения значения перешли 0 и стали слишком большими сбросить в 0 *)
		IF Buffer[3,i].a > 200 THEN
			Buffer[3,i].a:=0;
		END_IF
	END_FOR
	Turbo_Flag_minus_3:=FALSE;
END_IF
IF Turbo_Flag_minus_4 THEN
	FOR i:=1 TO 16 DO
		Buffer[4,i].a:=Buffer[4,i].a-Change_volume;
		(* Если из за уменьшения значения перешли 0 и стали слишком большими сбросить в 0 *)
		IF Buffer[4,i].a > 200 THEN
			Buffer[4,i].a:=0;
		END_IF
	END_FOR
	Turbo_Flag_minus_4:=FALSE;
END_IF
IF Turbo_Flag_minus_5 THEN
	FOR i:=1 TO 16 DO
		Buffer[5,i].a:=Buffer[5,i].a-Change_volume;
		(* Если из за уменьшения значения перешли 0 и стали слишком большими сбросить в 0 *)
		IF Buffer[5,i].a > 200 THEN
			Buffer[5,i].a:=0;
		END_IF
	END_FOR
	Turbo_Flag_minus_5:=FALSE;
END_IF
IF Turbo_Flag_minus_6 THEN
	FOR i:=1 TO 16 DO
		Buffer[6,i].a:=Buffer[6,i].a-Change_volume;
		(* Если из за уменьшения значения перешли 0 и стали слишком большими сбросить в 0 *)
		IF Buffer[6,i].a > 200 THEN
			Buffer[6,i].a:=0;
		END_IF
	END_FOR
	Turbo_Flag_minus_6:=FALSE;
END_IF
IF Turbo_Flag_minus_7 THEN
	FOR i:=1 TO 16 DO
		Buffer[7,i].a:=Buffer[7,i].a-Change_volume;
		(* Если из за уменьшения значения перешли 0 и стали слишком большими сбросить в 0 *)
		IF Buffer[7,i].a > 200 THEN
			Buffer[7,i].a:=0;
		END_IF
	END_FOR
	Turbo_Flag_minus_7:=FALSE;
END_IF
IF Turbo_Flag_minus_8 THEN
	FOR i:=1 TO 16 DO
		Buffer[8,i].a:=Buffer[8,i].a-Change_volume;
		(* Если из за уменьшения значения перешли 0 и стали слишком большими сбросить в 0 *)
		IF Buffer[8,i].a > 200 THEN
			Buffer[8,i].a:=0;
		END_IF
	END_FOR
	Turbo_Flag_minus_8:=FALSE;
END_IF

IF Turbo_Flag_minus_9 THEN
	FOR i:=1 TO 16 DO
		Buffer[9,i].a:=Buffer[9,i].a-Change_volume;
		(* Если из за уменьшения значения перешли 0 и стали слишком большими сбросить в 0 *)
		IF Buffer[9,i].a > 200 THEN
			Buffer[9,i].a:=0;
		END_IF
	END_FOR
	Turbo_Flag_minus_9:=FALSE;
END_IF
IF Turbo_Flag_minus_10 THEN
	FOR i:=1 TO 16 DO
		Buffer[10,i].a:=Buffer[10,i].a-Change_volume;
		(* Если из за уменьшения значения перешли 0 и стали слишком большими сбросить в 0 *)
		IF Buffer[10,i].a > 200 THEN
			Buffer[10,i].a:=0;
		END_IF
	END_FOR
	Turbo_Flag_minus_10:=FALSE;
END_IF
IF Turbo_Flag_minus_11 THEN
	FOR i:=1 TO 16 DO
		Buffer[11,i].a:=Buffer[11,i].a-Change_volume;
		(* Если из за уменьшения значения перешли 0 и стали слишком большими сбросить в 0 *)
		IF Buffer[11,i].a > 200 THEN
			Buffer[11,i].a:=0;
		END_IF
	END_FOR
	Turbo_Flag_minus_11:=FALSE;
END_IF
IF Turbo_Flag_minus_12 THEN
	FOR i:=1 TO 16 DO
		Buffer[12,i].a:=Buffer[12,i].a-Change_volume;
		(* Если из за уменьшения значения перешли 0 и стали слишком большими сбросить в 0 *)
		IF Buffer[12,i].a > 200 THEN
			Buffer[12,i].a:=0;
		END_IF
	END_FOR
	Turbo_Flag_minus_12:=FALSE;
END_IF
IF Turbo_Flag_minus_13 THEN
	FOR i:=1 TO 16 DO
		Buffer[13,i].a:=Buffer[13,i].a-Change_volume;
		(* Если из за уменьшения значения перешли 0 и стали слишком большими сбросить в 0 *)
		IF Buffer[13,i].a > 200 THEN
			Buffer[13,i].a:=0;
		END_IF
	END_FOR
	Turbo_Flag_minus_13:=FALSE;
END_IF
IF Turbo_Flag_minus_14 THEN
	FOR i:=1 TO 16 DO
		Buffer[14,i].a:=Buffer[14,i].a-Change_volume;
		(* Если из за уменьшения значения перешли 0 и стали слишком большими сбросить в 0 *)
		IF Buffer[14,i].a > 200 THEN
			Buffer[14,i].a:=0;
		END_IF
	END_FOR
	Turbo_Flag_minus_14:=FALSE;
END_IF
IF Turbo_Flag_minus_15 THEN
	FOR i:=1 TO 16 DO
		Buffer[15,i].a:=Buffer[15,i].a-Change_volume;
		(* Если из за уменьшения значения перешли 0 и стали слишком большими сбросить в 0 *)
		IF Buffer[15,i].a > 200 THEN
			Buffer[15,i].a:=0;
		END_IF
	END_FOR
	Turbo_Flag_minus_15:=FALSE;
END_IF
IF Turbo_Flag_minus_16 THEN
	FOR i:=1 TO 16 DO
		Buffer[16,i].a:=Buffer[16,i].a-Change_volume;
		(* Если из за уменьшения значения перешли 0 и стали слишком большими сбросить в 0 *)
		IF Buffer[16,i].a > 200 THEN
			Buffer[16,i].a:=0;
		END_IF
	END_FOR
	Turbo_Flag_minus_16:=FALSE;
END_IF
END_ACTION
ACTION Turbo_plus:
(* Добавляем фиксированное значение к текущему значению в столбце Turbo *)

IF Turbo_Flag_plus_1 THEN
	FOR i:=1 TO 16 DO
		Buffer[1,i].a:=Buffer[1,i].a+Change_volume;
	END_FOR
	Turbo_Flag_plus_1:=FALSE;
END_IF
IF Turbo_Flag_plus_2 THEN
	FOR i:=1 TO 16 DO
		Buffer[2,i].a:=Buffer[2,i].a+Change_volume;
	END_FOR
	Turbo_Flag_plus_2:=FALSE;
END_IF
IF Turbo_Flag_plus_3 THEN
	FOR i:=1 TO 16 DO
		Buffer[3,i].a:=Buffer[3,i].a+Change_volume;
	END_FOR
	Turbo_Flag_plus_3:=FALSE;
END_IF
IF Turbo_Flag_plus_4 THEN
	FOR i:=1 TO 16 DO
		Buffer[4,i].a:=Buffer[4,i].a+Change_volume;
	END_FOR
	Turbo_Flag_plus_4:=FALSE;
END_IF
IF Turbo_Flag_plus_5 THEN
	FOR i:=1 TO 16 DO
		Buffer[5,i].a:=Buffer[5,i].a+Change_volume;
	END_FOR
	Turbo_Flag_plus_5:=FALSE;
END_IF
IF Turbo_Flag_plus_6 THEN
	FOR i:=1 TO 16 DO
		Buffer[6,i].a:=Buffer[6,i].a+Change_volume;
	END_FOR
	Turbo_Flag_plus_6:=FALSE;
END_IF
IF Turbo_Flag_plus_7 THEN
	FOR i:=1 TO 16 DO
		Buffer[7,i].a:=Buffer[7,i].a+Change_volume;
	END_FOR
	Turbo_Flag_plus_7:=FALSE;
END_IF
IF Turbo_Flag_plus_8 THEN
	FOR i:=1 TO 16 DO
		Buffer[8,i].a:=Buffer[8,i].a+Change_volume;
	END_FOR
	Turbo_Flag_plus_8:=FALSE;
END_IF

IF Turbo_Flag_plus_9 THEN
	FOR i:=1 TO 16 DO
		Buffer[9,i].a:=Buffer[9,i].a+Change_volume;
	END_FOR
	Turbo_Flag_plus_9:=FALSE;
END_IF
IF Turbo_Flag_plus_10 THEN
	FOR i:=1 TO 16 DO
		Buffer[10,i].a:=Buffer[10,i].a+Change_volume;
	END_FOR
	Turbo_Flag_plus_10:=FALSE;
END_IF
IF Turbo_Flag_plus_11 THEN
	FOR i:=1 TO 16 DO
		Buffer[11,i].a:=Buffer[11,i].a+Change_volume;
	END_FOR
	Turbo_Flag_plus_11:=FALSE;
END_IF
IF Turbo_Flag_plus_12 THEN
	FOR i:=1 TO 16 DO
		Buffer[12,i].a:=Buffer[12,i].a+Change_volume;
	END_FOR
	Turbo_Flag_plus_12:=FALSE;
END_IF
IF Turbo_Flag_plus_13 THEN
	FOR i:=1 TO 16 DO
		Buffer[13,i].a:=Buffer[13,i].a+Change_volume;
	END_FOR
	Turbo_Flag_plus_13:=FALSE;
END_IF
IF Turbo_Flag_plus_14 THEN
	FOR i:=1 TO 16 DO
		Buffer[14,i].a:=Buffer[14,i].a+Change_volume;
	END_FOR
	Turbo_Flag_plus_14:=FALSE;
END_IF
IF Turbo_Flag_plus_15 THEN
	FOR i:=1 TO 16 DO
		Buffer[15,i].a:=Buffer[15,i].a+Change_volume;
	END_FOR
	Turbo_Flag_plus_15:=FALSE;
END_IF
IF Turbo_Flag_plus_16 THEN
	FOR i:=1 TO 16 DO
		Buffer[16,i].a:=Buffer[16,i].a+Change_volume;
	END_FOR
	Turbo_Flag_plus_16:=FALSE;
END_IF
END_ACTION

(* POU Ввод данных/Get_Currents, ST *)
PROGRAM Get_Currents
VAR
   fb_OutGetCurrent   : FB_x_out_get_current;
	s16_Return   	: INT;

	i,j,k: WORD; (* Счетчики количества аварийных событий *)
END_VAR
(******************* Контроль протекающего тока через выводы на обыв и короткое замыкание *************************************************************)

(* Контроль тока через газовые инжектора осуществляем только если они включены ( включен блок, имеется HOLD ток и не включен спец режим выключения гащза перед переключением на дизель )*)

IF Flag_ECU_ON AND Inj_PWM_time > 0 AND gq_Relay = TRUE		THEN

	Check_Inj1();
	Check_Inj2();
	Check_Inj3();

END_IF
END_PROGRAM
ACTION Check_Inj1:
	(* Находится ли ток через инжектор 1 в допустимых пределах ? *)
	(* Контроль по максимальным значениям не производится, так как ESX мериет максимальный ток с ошибкой *)
IF Flag_Inj1_ON AND  Inj_PWM_time > 0 AND Speed > p.Speed_limit THEN

	IF s32_Current_Inj1_1 < p.Min_inj_current OR s32_Current_Inj1_2 < p.Min_inj_current THEN
		i:=i+1;
	ELSE
		i:=0;
	END_IF

	(* Если ток инжектора 1 выходит задопустимые пределы Max_inj_current_time раз подряд, тогда ошибка *)
	IF i>=Max_inj_current_time THEN
		Err_Inj1:=TRUE;
		i:=Max_inj_current_time;					(* Что бы избежать переполнения и ложного сброса флага *)
	ELSE
		Err_Inj1:=FALSE;
	END_IF

END_IF
END_ACTION
ACTION Check_Inj2:
	(* Находится ли ток через инжектор 2 в допустимых пределах ? *)
	(* Контроль по максимальным значениям не производится, так как ESX мериет максимальный ток с ошибкой *)
IF Flag_Inj2_ON AND Inj_PWM_time > 0 AND Speed > p.Speed_limit THEN

	IF s32_Current_Inj2_1 < p.Min_inj_current OR s32_Current_Inj2_2 < p.Min_inj_current THEN
		j:=j+1;
	ELSE
		j:=0;
	END_IF

	(* Если ток инжектора 2 выходит задопустимые пределы Max_inj_current_time раз подряд, тогда ошибка *)
	IF j >= Max_inj_current_time THEN
		Err_Inj2:=TRUE;
		j:=Max_inj_current_time;					(* Что бы избежать переполнения и ложного сброса флага *)
	ELSE
		Err_Inj2:=FALSE;
	END_IF

END_IF
END_ACTION
ACTION Check_Inj3:
	(* Находится ли ток через инжектор 3 в допустимых пределах ? *)
	(* Контроль по максимальным значениям не производится, так как ESX мериет максимальный ток с ошибкой *)
IF Flag_Inj3_ON AND Inj_PWM_time > 0 AND Speed > p.Speed_limit THEN

	IF	s32_Current_Inj3_1 < p.Min_inj_current OR s32_Current_Inj3_2 < p.Min_inj_current THEN
		k:=k+1;
	ELSE
		k:=0;
	END_IF

	(* Если ток инжектора 3 выходит задопустимые пределы Max_inj_current_time раз подряд, тогда ошибка *)
	IF k >= Max_inj_current_time THEN
		Err_Inj3:=TRUE;
		k:=Max_inj_current_time;					(* Что бы избежать переполнения и ложного сброса флага *)
	ELSE
		Err_Inj3:=FALSE;
	END_IF

END_IF
END_ACTION

(* POU Ввод данных/Get_Reductor_press, ST *)
PROGRAM Get_Reductor_press
VAR
	s16_Return      				:INT;
   fb_InGetValue   				:FB_x_in_get_value;


END_VAR
fb_InGetValue(ou16_Channel:=X_IN_22, os32_Value=>Reductor_press, os16_Status=>s16_Return);

(* Находится ли давление в редукторе в допустимых пределах ? *)

IF Reductor_press < p.Min_Reductor_press THEN
		Count_min_reductor_press:=Count_min_reductor_press+1;
ELSE
	Count_min_reductor_press:=0;
END_IF

(* Если давление в редукторе выходит задопустимые пределы Reductor_press_time раз подряд, тогда ошибка *)
IF Count_min_reductor_press >= Min_Reductor_press_time THEN
		Err_Reductor_press:=TRUE;
		Count_min_reductor_press:=Min_Reductor_press_time;					(* Что бы избежать переполнения и ложного сброса флага *)
ELSE
		Err_Reductor_press:=FALSE;
END_IF
END_PROGRAM

(* POU Act_control, ST *)
PROGRAM Act_control
VAR
	TEST					:INT;

	x,y,z					:BYTE;  			(* Временные переменные, для определения ячейки калибровочной таблицы *)
	PPS_emul_cor		:DINT;			(* Добавочный поправочный коэффициент емуляции при резком нажатии на педаль газа *)
	s16_Return      	:INT;
   fb_InGetValue   	:FB_x_in_get_value;
	fb_OutSetValue  	:FB_x_out_set_value;
	PPS_PWM				:DINT:=800;		(* Используется в визуализации для ручного ввода уровня PWM при подборе *)
	Hold_manual			:BYTE; 			(* Значение Холда для ручного режима *)

(******** Check_PPS используются при проверки коррктности PPS **************************)
	PPS1_count			:WORD;			(* Счетчик количества циклов, когда PPS1 ошибочно *)
	PPS2_count			:WORD;			(* Счетчик количества циклов, когда PPS2 ошибочно *)
	PPS_ratio_count	:WORD;			(* Счетчик количества циклов, когда соотношение PPS1/PPS2 ошибочно *)
	PPS_ratio			:REAL;			(* Используется для вычисления соотношения PPS1 к PPS2 *)


END_VAR
(* Выбираем из калибровочной таблицы занчение желаемой подачи газа, соответствующее текущим оборотам, нагрузке и нажатию на педаль газа*)
fb_InGetValue(ou16_Channel:=X_IN_24, os32_Value=>PPS1, os16_Status=>s16_Return);
fb_InGetValue(ou16_Channel:=X_IN_25, os32_Value=>PPS2, os16_Status=>s16_Return);
(* Проверка допустимости значений PPS *)
Check_PPS();

x:=Get_TURBO_ARRAY_Number(Turbo_pressure);
y:=Get_RPM_ARRAY_Number(RPM);
z:=Get_Load_ARRAY_Number(Load);

(*******************************  Обработка режима эмуляции педали газа **********************************************************)

(* Если педаль хоть как-то нажата и набрана скорость, то вычислять подачу дизеля*)
IF PPS1 >= p.PPS_table[2]  AND Speed > p.Speed_limit THEN
	PPS1_emul:= PPS1 - (10*p.Cal_table[ x,y ].DIESEL)*(PPS1*100/p.PPS_table[16]) /100;
	PPS1_emul:=PPS1_emul-p.DIESEL_Load_table[z];
ELSE
	PPS1_emul:= PPS1;
END_IF

Check_PPS_emul(); (* Проверка допустимости полученного сигнала эмуляции PPS *)
Put_PPS_emul();	(* Выдача сиганала эмуляции PPS *)

(* Если не режим тестирования инжекторов с ручным заданием значения HOLD *)
IF Flag_test_inj=FALSE THEN
	(* Если педаль хоть как-то нажата, то вычислять подачу газа*)
	IF PPS1 >= p.PPS_table[2] AND Speed > p.Speed_limit THEN
		(* Установка длительности выдачи газа, автоматический рабочий режим *)
		Hold_time:=DINT_TO_BYTE((p.Cal_table[ x,y ].GAS*(PPS1*100/p.PPS_table[16]))/100);
		Hold_time:=INT_TO_BYTE(BYTE_TO_INT(Hold_time)-p.GAS_Load_table[z]);
		TEST:=p.GAS_Load_table[z];
		EGT_correction();	(* Коррекция холда по EGT *)
		IF Flag_24V THEN  (* Если система с 24 В форсунками, то используем спецкоды для уменьшения подачи *)
			Special_code();		(* Обработка спецкодов, для уменьшения подачи *)
		ELSE
			Inj_PWM_time:=Hold_time;	(* Если нет спецкодов, то просто холд из таблицы *)
		END_IF
		Inj_PWM_time:=Inj_PWM_time*4;  (* Переводим в циклы по 250 мкс *)
	ELSE
		Inj_PWM_time:=0;     (* Если педаль газа не нажата *)
		Hold_time:=0;
	END_IF
ELSE
	(* Установка длительности выдачи газа, ручной настроечный режим *)
	Inj_PWM_time:=Hold_manual*4;
END_IF

(****************** Проверки выполняются в любом случае ********************************************)

Flag_Inj_PWM_cor:=FALSE;

(* Ограничение предельного значения холда, в том числе особо жесткое на маленьких оборотах и надувах *)
	IF RPM < p.RPM_table[3] AND Turbo_pressure < p.Turbo_table[3] AND Inj_PWM_time > p.Inj_MAX_hold_time_min THEN
		Inj_PWM_time:=p.Inj_MAX_hold_time_min;
		Flag_Inj_PWM_cor:=TRUE;
	ELSIF Inj_PWM_time > p.Inj_MAX_hold_time THEN
		Inj_PWM_time:=p.Inj_MAX_hold_time;
		Flag_Inj_PWM_cor:=TRUE;
	END_IF
END_PROGRAM
ACTION Check_PPS:
(* Проверка допустимости значений PPS *)

(* Если PPS1, PPS2 и их соотношение  не попадает в заданые пределы уже более PPS_err_time раз *)

(* Находится ли PPS1 в допустимых пределах ? *)
IF PPS1 < p.PPS1_min OR PPS1 > p.PPS1_max THEN
		PPS1_count:=PPS1_count+1;
		IF PPS1_count > PPS_err_time THEN
			Err_PPS:=TRUE;
		END_IF
ELSE
	PPS1_count:=0;
END_IF

(* Находится ли PPS2 в допустимых пределах ? *)
IF PPS2 < p.PPS2_min OR PPS2 > p.PPS2_max THEN
		PPS2_count:=PPS2_count+1;
		IF PPS2_count > PPS_err_time THEN
			Err_PPS:=TRUE;
		END_IF
ELSE
	PPS2_count:=0;
END_IF

PPS_ratio:=DINT_TO_REAL(PPS1)/DINT_TO_REAL(PPS2);

(* Находится ли соотношение PPS1/PPS2 в допустимых пределах ? *)
IF PPS_ratio < p.PPS_ratio_min OR PPS_ratio > p.PPS_ratio_max THEN
		PPS_ratio_count:=PPS_ratio_count+1;
		IF PPS_ratio_count > PPS_err_time THEN
			Err_PPS:=TRUE;
		END_IF
ELSE
	PPS_ratio_count:=0;
END_IF
END_ACTION
ACTION Check_PPS_emul:
(* Проверка, что бы эмуляция не выходила за границы возможного физического диапазона *)
IF PPS1_emul < p.PPS1_min THEN
			PPS1_emul:=p.PPS_table[1];
END_IF

IF PPS1_emul > p.PPS1_max THEN
		PPS1_emul:=p.PPS_table[16];
END_IF
END_ACTION
ACTION EGT_correction:
(*
		CASE EGT OF
			0..2600: Hold_time:=Hold_time-13;
			2601..2700:  Hold_time:=Hold_time-12;
			2701..2800:  Hold_time:=Hold_time-11;
			2801..2900:  Hold_time:=Hold_time-10;
			2901..3000:  Hold_time:=Hold_time-9;
			3001..3100:  Hold_time:=Hold_time-8;
			3101..3200:  Hold_time:=Hold_time-7;
			3201..3300:  Hold_time:=Hold_time-6;
			3301..3400:  Hold_time:=Hold_time-5;
			3401..3500:  Hold_time:=Hold_time-4;
			3501..3600:  Hold_time:=Hold_time-3;
			3601..3700:  Hold_time:=Hold_time-2;
			3701..3800:  Hold_time:=Hold_time-1;
		END_CASE
		IF hold_time > 40 THEN
			Hold_time:=0;
		END_IF
*)
;
END_ACTION
ACTION Put_PPS_emul:
(* Если не включен режим исследования зависимости PWM и выхода напряжения с операционного усилителя, то выдаем значения PWM из таблицы соответствия PWM напряжению *)
IF Flag_PWM_researh THEN
	(* Выдача PWM на операционник для эмуляции PPS, уровень PWM получен в ручном режиме из визуализации *)
	fb_OutSetValue(ou16_Channel:=X_OUT_04, os32_Value:=PPS_PWM, os16_Status=>s16_Return);
ELSE
	(* Выборка уровня PWM для выдачи на операционный усилитель для емуляции PPS1 *)
	PPS_PWM:=p.PPS1_emul_PWM[Get_PPS_ARRAY_Number(PPS1_emul)];
	(* Выдача PWM на операционник для эмуляции PPS *)
	fb_OutSetValue(ou16_Channel:=X_OUT_04, os32_Value:=PPS_PWM, os16_Status=>s16_Return);
END_IF
END_ACTION
ACTION Special_code:
(* 1 и 2 - спецкоды, применяются для отключения форсунок с целью уменьшения подачи *)
			CASE HOLD_time OF
				1: 	Inj_PWM_time:=4;			(* Работает только третий инжектор *)
						Flag_Inj1_ON:=FALSE;
						Flag_Inj2_ON:=FALSE;
						Flag_Inj3_ON:=TRUE;
				2:
						Inj_PWM_time:=4;			(* Работает только первый и второй инжектор *)
						Flag_Inj3_ON:=FALSE;
						Flag_Inj1_ON:=TRUE;
						Flag_Inj2_ON:=TRUE;
			ELSE
				(* Восстанавливаем в рабочее состояние инжектора, возможно отключенные спецкодами 71 и 72 *)
				Flag_Inj1_ON:=TRUE;
				Flag_Inj2_ON:=TRUE;
				Flag_Inj3_ON:=TRUE;

				(*** ВАЖНО ! Из-за спецкодов отключения 1 и 2 форсунок для малой подачи все калибровочный таблицы сдвигаются на 2 влево 3=1, 4=2 и т.д*)
				IF HOLD_time > 2 THEN
					Inj_PWM_time:=HOLD_time-2;
				ELSE
					Inj_PWM_time:=0;
					Flag_Inj1_ON:=FALSE;
					Flag_Inj2_ON:=FALSE;
					Flag_Inj3_ON:=FALSE;
				END_IF
			END_CASE
END_ACTION

(* POU Выборка значения из массива/Get_TURBO_ARRAY_Number, ST *)
FUNCTION Get_TURBO_ARRAY_Number : BYTE
VAR_INPUT
	Turbo_now:DINT;
END_VAR
VAR
	i:BYTE:=1;
	j:BYTE:=16;
	med:BYTE;
END_VAR
(* Функция в качестве аргумента принимает, давление надува в мВольтах, а возвращает номер элемента массива, соответствующего этому количеству оборотов *)


(* Делим массив каждый раз пополам, проверяя где находится искомый элемент, пока границы массива не сойдутся*)

WHILE i<>j  DO
	med:=(i+j)/2;
	IF TURBO_now>p.TURBO_table[med] THEN
		i:=med+1;
	ELSE
		j:=med;
	END_IF
END_WHILE


Get_TURBO_ARRAY_Number :=i;							(* Номер , когда границы сошлись и совпадают с краями массива не нуждается в уточнении *)

(* Уточняем какой элемент массива наиболее сответствует, кол-ву оборотов переданному как элемент функции *)
(* определяем спава или слева от найдено индекса находится ребуемый элемент и в зависмимости от этого действеум *)

IF i=med AND i<>1 THEN
	IF ABS(p.TURBO_table[med-1]-TURBO_now)<= ABS(p.TURBO_table[med]-TURBO_now) THEN
		Get_TURBO_ARRAY_Number :=med-1;
	ELSE
		Get_TURBO_ARRAY_Number :=med;
	END_IF
ELSIF i<>med AND  i<>16 THEN
	IF ABS(p.TURBO_table[med+1]-TURBO_now)<= ABS(p.TURBO_table[med]-TURBO_now) THEN
		Get_TURBO_ARRAY_Number :=med+1;
	ELSE
		Get_TURBO_ARRAY_Number :=med;
	END_IF
END_IF
END_FUNCTION

(* POU Выборка значения из массива/Get_RPM_ARRAY_Number, ST *)
FUNCTION Get_RPM_ARRAY_Number : BYTE
VAR_INPUT
	RPM_now:DINT;
END_VAR
VAR
	i:BYTE:=1;
	j:BYTE:=16;
	med:BYTE;
END_VAR
(* Функция в качестве аргумента принимает, количество оборотов, а возвращает номер элемента массива, соответствующего этому количеству оборотов *)


(* Делим массив каждый раз пополам, проверяя где находится искомый элемент, пока границы массива не сойдутся*)

WHILE i<>j  DO
	med:=(i+j)/2;
	IF RPM_now>p.RPM_table[med] THEN
		i:=med+1;
	ELSE
		j:=med;
	END_IF
END_WHILE


Get_RPM_ARRAY_Number :=i;							(* Номер , когда границы сошлись и совпадают с краями массива не нуждается в уточнении *)

(* Уточняем какой элемент массива наиболее сответствует, кол-ву оборотов переданному как элемент функции *)
(* определяем спава или слева от найдено индекса находится ребуемый элемент и в зависмимости от этого действеум *)

IF i=med AND i<>1 THEN
	IF ABS(p.RPM_table[med-1]-RPM_now)<= ABS(p.RPM_table[med]-RPM_now) THEN
		Get_RPM_ARRAY_Number :=med-1;
	ELSE
		Get_RPM_ARRAY_Number :=med;
	END_IF
ELSIF i<>med AND  i<>16 THEN
	IF ABS(p.RPM_table[med+1]-RPM_now)<= ABS(p.RPM_table[med]-RPM_now) THEN
		Get_RPM_ARRAY_Number :=med+1;
	ELSE
		Get_RPM_ARRAY_Number :=med;
	END_IF
END_IF
END_FUNCTION

(* POU Выборка значения из массива/Get_Load_ARRAY_Number, ST *)
FUNCTION Get_Load_ARRAY_Number : BYTE
VAR_INPUT
	Load_now:DINT;
END_VAR
VAR
	i:BYTE:=1;
	j:BYTE:=16;
	med:BYTE;
END_VAR
(* Функция в качестве аргумента принимает, количество оборотов, а возвращает номер элемента массива, соответствующего этому количеству оборотов *)


(* Делим массив каждый раз пополам, проверяя где находится искомый элемент, пока границы массива не сойдутся*)

WHILE i<>j  DO
	med:=(i+j)/2;
	IF Load_now>p.Load_table[med] THEN
		i:=med+1;
	ELSE
		j:=med;
	END_IF
END_WHILE


Get_Load_ARRAY_Number :=i;							(* Номер , когда границы сошлись и совпадают с краями массива не нуждается в уточнении *)

(* Уточняем какой элемент массива наиболее сответствует, кол-ву оборотов переданному как элемент функции *)
(* определяем спава или слева от найдено индекса находится ребуемый элемент и в зависмимости от этого действеум *)

IF i=med AND i<>1 THEN
	IF ABS(p.Load_table[med-1]-Load_now)<= ABS(p.Load_table[med]-Load_now) THEN
		Get_Load_ARRAY_Number :=med-1;
	ELSE
		Get_Load_ARRAY_Number :=med;
	END_IF
ELSIF i<>med AND  i<>16 THEN
	IF ABS(p.Load_table[med+1]-Load_now)<= ABS(p.Load_table[med]-Load_now) THEN
		Get_Load_ARRAY_Number :=med+1;
	ELSE
		Get_Load_ARRAY_Number :=med;
	END_IF
END_IF
END_FUNCTION

(* POU Выборка значения из массива/Get_PPS_ARRAY_Number, ST *)
FUNCTION Get_PPS_ARRAY_Number : BYTE
VAR_INPUT
	PPS_now:DINT;
END_VAR
VAR
	i:BYTE:=1;
	j:BYTE:=16;
	med:BYTE;
END_VAR
(* Функция в качестве аргумента принимает, PPS, а возвращает номер элемента массива, соответствующего этому PPS *)

(* Делим массив каждый раз пополам, проверяя где находится искомый элемент, пока границы массива не сойдутся*)

WHILE i<>j  DO
	med:=(i+j)/2;
	IF PPS_now>p.PPS_table[med] THEN
		i:=med+1;
	ELSE
		j:=med;
	END_IF
END_WHILE


Get_PPS_ARRAY_Number :=i;							(* Номер , когда границы сошлись и совпадают с краями массива не нуждается в уточнении *)

(* Уточняем какой элемент массива наиболее сответствует, кол-ву оборотов переданному как элемент функции *)
(* определяем спава или слева от найдено индекса находится ребуемый элемент и в зависмимости от этого действеум *)

IF i=med AND i<>1 THEN
	IF ABS(p.PPS_table[med-1]-PPS_now)<= ABS(p.RPM_table[med]-PPS_now) THEN
		Get_PPS_ARRAY_Number :=med-1;
	ELSE
		Get_PPS_ARRAY_Number :=med;
	END_IF
ELSIF i<>med AND  i<>16 THEN
	IF ABS(p.PPS_table[med+1]-PPS_now)<= ABS(p.PPS_table[med]-PPS_now) THEN
		Get_PPS_ARRAY_Number :=med+1;
	ELSE
		Get_PPS_ARRAY_Number :=med;
	END_IF
END_IF
END_FUNCTION

(* POU Ввод данных/Get_Turbo, ST *)
PROGRAM Get_Turbo
VAR
	s16_Return      : INT;
   fb_InGetValue   : FB_x_in_get_value;
END_VAR
fb_InGetValue(ou16_Channel:=X_IN_21, os32_Value=>Turbo_pressure, os16_Status=>s16_Return);
END_PROGRAM

(* POU Ввод данных/Get_Key, ST *)
PROGRAM Get_Key
VAR
	s16_Return      : INT;
   fb_InGetValue   : FB_x_in_get_value;

	DF_switch	:DINT;
	DF_flag		:BOOL;

END_VAR
fb_InGetValue(ou16_Channel:=X_IN_12, os32_Value=>DF_switch, os16_Status=>s16_Return);

IF DF_switch=0 THEN					(* Если конпока изменения режима работы ECU нажата, то...*)
	IF DF_flag THEN					(* Первый ли цикл когда она нажата ? *)
		DF_flag:=FALSE;				(*Выставляем флажок, для  игнорирования этой ветви, до тех пор пока кнопка не изменит своего положения *)
		IF Flag_ECU_ON THEN			(* Включаем или выключаем газодизельный режим ECU*)
			Flag_ECU_ON:=FALSE;
		ELSE
			Flag_ECU_ON:=TRUE;
			Count_min_reductor_press:=0; (* При переключении режимов начать отчет времени когда далвение было минимальным с 0 *)
		END_IF;
	END_IF
ELSE
	DF_flag:=TRUE;				(* Кнопка была отпущена, устанвкливаем разрешительный флажок для обработки следующего нажатия *)
END_IF
END_PROGRAM

(* POU Ввод данных/Get_Gas_meter, ST *)
PROGRAM Get_Gas_meter
VAR
	s16_Return      : INT;
   fb_InGetValue   : FB_x_in_get_value;
	fb_OutSetValue   : FB_x_out_set_value;

	i: DINT;
END_VAR
(* Считать значениедатчика кол-ва газа *)
fb_InGetValue(ou16_Channel:=X_IN_19, os32_Value=>Gas_meter, os16_Status=>s16_Return);

(* Определить уровень PWM для зажигания LED *)
i:=p.LED_BAR_PWM[Get_Gas_meter_ARRAY_Number(Gas_meter)];

(* Выдать PWM на LED bar *)
fb_OutSetValue(ou16_Channel:=X_OUT_03, os32_Value:=i, os16_Status=>s16_Return);
END_PROGRAM

(* POU Выборка значения из массива/Get_Gas_meter_ARRAY_Number, ST *)
FUNCTION Get_Gas_meter_ARRAY_Number : BYTE
VAR_INPUT
	Gas_meter_now:DINT;
END_VAR
VAR
	i:BYTE:=1;
	j:BYTE:=5;
	med:BYTE;
	Gas_meter_volume: BOOL;
END_VAR
(* Функция в качестве аргумента принимает, количество оборотов, а возвращает номер элемента массива, соответствующего этому PPS *)


(* Делим массив каждый раз пополам, проверяя где находится искомый элемент, пока границы массива не сойдутся*)

WHILE i<>j  DO
	med:=(i+j)/2;
	IF Gas_meter_now>p.Gas_meter_volume[med] THEN
		i:=med+1;
	ELSE
		j:=med;
	END_IF
END_WHILE


Get_Gas_meter_ARRAY_Number :=i;							(* Номер , когда границы сошлись и совпадают с краями массива не нуждается в уточнении *)

(* Уточняем какой элемент массива наиболее сответствует, кол-ву оборотов переданному как элемент функции *)
(* определяем спава или слева от найдено индекса находится ребуемый элемент и в зависмимости от этого действеум *)

IF i=med AND i<>1 THEN
	IF ABS(p.Gas_meter_volume[med-1]-Gas_meter_now)<= ABS(p.Gas_meter_volume[med]-Gas_meter_now) THEN
		Get_Gas_meter_ARRAY_Number :=med-1;
	ELSE
		Get_Gas_meter_ARRAY_Number :=med;
	END_IF
ELSIF i<>med AND  i<>16 THEN
	IF ABS(p.Gas_meter_volume[med+1]-Gas_meter_now)<= ABS(p.Gas_meter_volume[med]-Gas_meter_now) THEN
		Get_Gas_meter_ARRAY_Number :=med+1;
	ELSE
		Get_Gas_meter_ARRAY_Number :=med;
	END_IF
END_IF
END_FUNCTION

(* POU Ввод данных/Get_Reductor_temp, ST *)
PROGRAM Get_Reductor_temp
VAR
	s16_Return      : INT;
   fb_InGetValue   : FB_x_in_get_value;

	(* Температура редуктора уже в норме, время до следующей проверки пошло *)
	Flag_Err_Reductor_temp: BOOL;
	(* Счетчик циклов до следующей проверки *)
	Count_max_Reductor_temp: WORD;

END_VAR
fb_InGetValue(ou16_Channel:=X_IN_20, os32_Value=>Reductor_temp, os16_Status=>s16_Return);

(* Если температура редуктора превысила допустимую температуру для включения, то следующий
контроль произойдет через некоторое время,что бы избежать дребезга *)

IF Flag_Err_Reductor_temp AND  Count_max_Reductor_temp < Reductor_temp_err_time THEN
	Count_max_reductor_temp:=Count_max_reductor_temp+1;
ELSE
	Count_max_Reductor_temp:=0;
	(* Находится ли температура редуктора в допустимых пределах ? *)
	IF Reductor_temp < p.Reductor_temp_work THEN
		Flag_Err_Reductor_temp:=TRUE;
		Err_Reductor_temp:=TRUE;
	ELSE
		Flag_Err_Reductor_temp:=FALSE;
		Err_Reductor_temp:=FALSE;
	END_IF
END_IF
END_PROGRAM

(* POU Ввод данных/Get_Inj_temp, ST *)
PROGRAM Get_Inj_temp
VAR
	s16_Return      : INT;
   fb_InGetValue   : FB_x_in_get_value;
END_VAR
fb_InGetValue(ou16_Channel:=X_IN_15, os32_Value=>Injector_temp, os16_Status=>s16_Return);

(* Находится ли температура форсунок в допустимых пределах ? *)
(* Если температура форсунок хоть один раз превысила допустимый порог, то снять ошибку можно только перегрузкой *)

IF Injector_temp > p.Inj_temp_max THEN
	Err_inj_temp:=TRUE;
END_IF
END_PROGRAM

(* POU Ввод данных/Get_FUEL_meter, ST *)
PROGRAM Get_FUEL_meter
VAR
	s16_Return      : INT;
   fb_InGetValue   : FB_x_in_get_value;
	fb_OutSetValue   : FB_x_out_set_value;
	q: WORD;
END_VAR
(* Считать значениедатчика кол-ва солярки *)
fb_InGetValue(ou16_Channel:=X_IN_18, os32_Value=>FUEL_meter, os16_Status=>s16_Return);
(*Взять из таблицы физическое згачение объема слоответствующее показанию датчика *)
q:= p.FUEL_meter_liter[ Get_FUEL_meter_ARRAY_Number(FUEL_meter)];
FUEL_volume:=DINT_TO_REAL(FUEL_meter) * WORD_TO_REAL( q );
IF p.FUEL_meter_dat[Get_FUEL_meter_ARRAY_Number(FUEL_meter)] <> 0 THEN
	FUEL_volume:=FUEL_volume/WORD_TO_REAL(p.FUEL_meter_dat[Get_FUEL_meter_ARRAY_Number(FUEL_meter)]);
END_IF
END_PROGRAM

(* POU Выборка значения из массива/Get_FUEL_meter_ARRAY_Number, ST *)
FUNCTION Get_FUEL_meter_ARRAY_Number : BYTE
VAR_INPUT
	FUEL_meter_now:DINT;
END_VAR
VAR
	i:BYTE:=1;
	j:BYTE:=32;
	med:BYTE;
	FUEL_meter_dat: BOOL;
END_VAR
(* Функция в качестве аргумента принимает, количество оборотов, а возвращает номер элемента массива, соответствующего этому PPS *)


(* Делим массив каждый раз пополам, проверяя где находится искомый элемент, пока границы массива не сойдутся*)

WHILE i<>j  DO
	med:=(i+j)/2;
	IF FUEL_meter_now>p.FUEL_meter_dat[med] THEN
		i:=med+1;
	ELSE
		j:=med;
	END_IF
END_WHILE


Get_FUEL_meter_ARRAY_Number :=i;							(* Номер , когда границы сошлись и совпадают с краями массива не нуждается в уточнении *)

(* Уточняем какой элемент массива наиболее сответствует, кол-ву оборотов переданному как элемент функции *)
(* определяем спава или слева от найдено индекса находится ребуемый элемент и в зависмимости от этого действеум *)

IF i=med AND i<>1 THEN
	IF ABS(p.FUEL_meter_dat[med-1]-FUEL_meter_now)<= ABS(p.FUEL_meter_dat[med]-FUEL_meter_now) THEN
		Get_FUEL_meter_ARRAY_Number :=med-1;
	ELSE
		Get_FUEL_meter_ARRAY_Number :=med;
	END_IF
ELSIF i<>med AND  i<>32 THEN
	IF ABS(p.FUEL_meter_dat[med+1]-FUEL_meter_now)<= ABS(p.FUEL_meter_dat[med]-FUEL_meter_now) THEN
		Get_FUEL_meter_ARRAY_Number :=med+1;
	ELSE
		Get_FUEL_meter_ARRAY_Number :=med;
	END_IF
END_IF
END_FUNCTION

(* POU Ввод данных/Get_cPPS, ST *)
PROGRAM Get_cPPS
VAR
	fb_InGetValue   : FB_x_in_get_value;
	s16_Return      : INT;
END_VAR
(* Взяьть реальное значение выдаваемого напряжения эмуляции PPS *)
fb_InGetValue(ou16_Channel:=X_IN_26, os32_Value=>cPPS1_emul, os16_Status=>s16_Return);
END_PROGRAM

(* POU CAN/Send, ST *)
PROGRAM Send
VAR
	s16_Return       		: INT;
	t_Msg             	: T_x_can_msg;
   fb_CanObjSendMsg   	: FB_x_can_obj_send_msg;
	fb_EepRead  			: FB_x_eep_read;
	u16_Crc           	: UINT;
	fb_UtiCalcCrc16   	: FB_x_uti_calc_crc_16;
	CAN_TX_count			:WORD:=10000;				(* Счетчик переданных пакетов по CAN *)

END_VAR
IF Flag_CAN THEN

	IF Flag_CAN_Write THEN
		Flag_CAN_Write:=FALSE;
		t_Msg.t_Id.u32_Id := 16#101;
		t_Msg.t_Id.u8_Xtd := 0;
		t_Msg.u8_Dlc      := 8;				(* Количество передаваемых байт *)
		t_Msg.au8_Data[0] := 1;
		t_Msg.au8_Data[1] := 9;
		t_Msg.au8_Data[2] := 7;
		t_Msg.au8_Data[3] := 2;
		t_Msg.au8_Data[4] := 1;
		t_Msg.au8_Data[5] := 9;
		t_Msg.au8_Data[6] := 7;
		t_Msg.au8_Data[7] := 2;
		fb_CanObjSendMsg(ou32_Handle:=TX, ot_Msg:=t_Msg, os16_Status=>s16_Return);
	END_IF


	IF Flag_CAN_send THEN											(* Первоначальная процедура, выполняется один раз по команде от Питоновской программе *)
		(* Читаем все содержимое энергонезависимой памяти *)
		fb_EepRead(ou32_Address:=0, ou32_Count:=SIZEOF(Can_buffer), opu8_Data:=ADR(Can_buffer), os16_Status=>s16_Return);
		(* Вычисляем CRC16 для массива передаваемых данных *)
		u16_Crc:=16#1D0F;
		fb_UtiCalcCrc16(ou32_Count:=SIZEOF(Can_buffer)-2, opu8_Data:=ADR(Can_buffer), ou16_Crc:=u16_Crc, os16_Status=>s16_Return);
		Can_buffer[SIZEOF(Can_buffer)-1]:=WORD_TO_BYTE(u16_Crc);
		Can_buffer[SIZEOF(Can_buffer)]:=WORD_TO_BYTE(u16_Crc/256);
		CAN_TX_count:=0;
		Flag_CAN_send:=FALSE;


	ELSIF CAN_TX_count <=  (SIZEOF(Can_buffer)-8) THEN						(* Передача основных данных, выполняется 1 раз после хандшейка *)

